# B&R Automation Studio project 8238 (part 6)

#### _config.st - *Read/Write Config Data
```iecst
ACTION _config:

	state 		ACCESS ADR(fuse.Internal.config_state);
	read_8		ACCESS ADR(fuse.Functions.Read_8);
	read_16		ACCESS ADR(fuse.Functions.Read_16);
	write		ACCESS ADR(fuse.Functions.Write);
	error		ACCESS ADR(fuse.Internal.LastError);

	read_8.pDeviceName 		:= fuse.pDevice;
	read_8.pData			:= ADR(fuse.Internal.Data_8);
	read_8.datatype 		:= ioLinkTYPE_USINT;
	read_8.dataLen			:= SIZEOF(fuse.Internal.Data_8);
	read_8.subIndex 		:= 0;

	read_16.pDeviceName 	:= fuse.pDevice;
	read_16.pData			:= ADR(fuse.Internal.Data_16);
	read_16.datatype 		:= ioLinkTYPE_UINT;
	read_16.dataLen			:= SIZEOF(fuse.Internal.Data_16);
	read_16.subIndex 		:= 0;

	write.pDeviceName := fuse.pDevice;
	write.pData 	:= ADR(fuse.Internal.WriteData);

	CASE state OF
		0:// Init  Turn of all functions just in case.
			fuse.Info.CommsOk := 0;
			state := 1;

		1://
			read_8.enable 	:= 0;
			read_8();
			IF (read_8.status = ERR_FUB_ENABLE_FALSE) THEN
				state := 2;
			END_IF;

		2:
			read_16.enable 	:= 0;
			read_16();
			IF (read_16.status = ERR_FUB_ENABLE_FALSE) THEN
				state := 3;
			END_IF;

		3..9:
			write.enable := 0;
			write();
			IF (write.status = ERR_FUB_ENABLE_FALSE) THEN
				state := 10;
			END_IF;

		10://Read the number of nodes.
			read_8.enable 	:= 1;
			read_8.index		:= 91;
			read_8();
			IF (read_8.status = ERR_OK) THEN
				fuse.Info.CommsOk := 1;
				fuse.Info.NoNodes := fuse.Internal.Data_8;
				fuse.Internal.Data_8 := 0;
				IF (fuse.Info.NoNodes > 0) THEN
					IF fuse.Info.NoNodes > MAX_FUSE_CHANNELS THEN
						fuse.Info.NoNodes := MAX_FUSE_CHANNELS;
					END_IF;
					state := 11;
				ELSE
					state := 0;
				END_IF;
			ELSIF (read_8.status <> ERR_FUB_BUSY) AND (read_8.status <> ERR_FUB_ENABLE_FALSE)  THEN  // Error read_8ing re initialise
				error := read_8.status;
				fuse.Info.CommsOk := 0;
				state := 0;
			END_IF;

		11..50:// read_8 the type  MAX 40 Fuses.
			channel := (state - 10);
			IF channel <= fuse.Info.NoNodes THEN
				read_8.enable 	:= 1;
				read_8.index		:= 900 + channel;
				read_8();
				IF (read_8.status = ERR_OK) THEN
					fuse.Info.Channel[channel].Type := fuse.Internal.Data_8;
					state := state + 1;
				ELSIF (read_8.status <> ERR_FUB_BUSY) AND (read_8.status <> ERR_FUB_ENABLE_FALSE)  THEN  // Error read_8ing re initialise
					fuse.Info.CommsOk := 0;
					state := 0;
				END_IF;
			ELSE
				state := 51;
			END_IF;

		51..90:// read_8 the trip current
			channel := (state - 50);
			IF channel <= fuse.Info.NoNodes THEN
				read_8.enable 	:= 1;
				read_8.index		:= 400 + channel;
				read_8();
				IF (read_8.status = ERR_OK) THEN
					fuse.Info.CommsOk := 1;
					fuse.Info.Channel[channel].TripCurrent := fuse.Internal.Data_8;
					state := state + 1;
				ELSIF (read_8.status <> ERR_FUB_BUSY) AND (read_8.status <> ERR_FUB_ENABLE_FALSE)  THEN  // Error reading re initialise
					state := 0;
				END_IF;
			ELSE
				state := 91;
			END_IF;

		91://Release the function block
			read_8.enable := 0;
			read_8();
			IF (read_8.status = ERR_FUB_ENABLE_FALSE) THEN
				state := 92;
			END_IF;

		92..93: // Read the max voltage
			read_16.enable := 1;
			read_16.datatype := ioLinkTYPE_INT;
			read_16.index		:= 100;
			read_16();
			IF (read_16.status = ERR_OK) THEN
				fuse.Info.CommsOk := 1;
				fuse.Info.MaxVoltage := fuse.Internal.Data_16;
				state := state + 1;
			ELSIF (read_16.status <> ERR_FUB_BUSY) AND (read_16.status <> ERR_FUB_ENABLE_FALSE)  THEN  // Error read_16ing re initialise
				fuse.Info.CommsOk := 0;
				state := 0;
			END_IF;

		94:// Read the Min Voltage;
			read_16.enable 	:= 1;
			read_16.datatype := ioLinkTYPE_INT;
			read_16.index		:= 101;
			read_16();
			IF (read_16.status = ERR_OK) THEN
				fuse.Info.CommsOk := 1;
				fuse.Info.MinVoltage :=  fuse.Internal.Data_16;
				state := state + 1;
			ELSIF (read_16.status <> ERR_FUB_BUSY) AND (read_16.status <> ERR_FUB_ENABLE_FALSE)  THEN  // Error reading re initialise
				fuse.Info.CommsOk := 0;
				state := 0;
			END_IF;

		95..100: // Disable the 16 way
			read_16.enable := 0;
			read_16();
			IF (read_16.status = ERR_FUB_ENABLE_FALSE) THEN
				state := 101;
			END_IF;

		101..140: // Read the channel status
			channel := (state - 100);
			IF channel <= fuse.Info.NoNodes THEN
				read_8.enable := 1;
				read_8.index := 500 + channel;
				read_8();
				IF (read_8.status = ERR_OK) THEN
					fuse.Info.Channel[channel].Status := fuse.Internal.Data_8;
					state := state + 1;
				END_IF;
			ELSE
				state := 141;
			END_IF;

		141: // Decide what to do next?
			//Check for differences then write if required
			//Check if the Min voltage has changed.
			IF (fuse.Info.MinVoltage <> fuse.Settings.MinVoltage) AND (fuse.Settings.MinVoltage > 0) THEN
				state := 150;
			END_IF;
			//Check if the Max voltage has changed.
			IF (fuse.Info.MaxVoltage <> fuse.Settings.MaxVoltage) AND (fuse.Settings.MaxVoltage > 0) THEN
				state := 151;
			END_IF;
			IF (fuse.Info.NoNodes > 0) THEN
				// Check if the trip current has changed
				FOR n := 1 TO fuse.Info.NoNodes DO
					IF (fuse.Info.Channel[n].TripCurrent <> fuse.Settings.Channel[n].TripCurrent) AND (fuse.Settings.Channel[n].TripCurrent > 0) THEN
						state := 161;
						EXIT;
					END_IF;
				END_FOR;
				// Check if the state has changed
				FOR n := 1 TO fuse.Info.NoNodes DO
					CASE fuse.Info.Channel[n].Status  OF
						EB_STATE_NC, EB_STATE_TRIP_SW_OFF:  // We cannot do anything is software.
							// We can;t do anything.

						EB_STATE_ON,EB_STATE_I_90, EB_STATE_I_100:
							IF (fuse.Settings.Channel[n].SetState = EB_SET_STATE_OFF ) THEN
								state := 200 + n;
								EXIT;
							END_IF;

						EB_STATE_TRIP, EB_STATE_TRIP_THERMAL, EB_STATE_TRIP_HARDWARE:
							IF (fuse.Settings.Channel[n].SetState = EB_SET_STATE_RESET ) THEN
								state := 200 + n;
								EXIT;
							END_IF;

						EB_STATE_OFF: // Turned off by hand
							IF (fuse.Settings.Channel[n].SetState = EB_SET_STATE_ON ) THEN
								state := 200 + n;
								EXIT;
							END_IF;
					END_CASE;
					IF (state = 141) THEN
						fuse.Settings.Channel[n].SetState := 0;	// Setting is not valid and cannot be actioned so clear it.
					END_IF;
				END_FOR;

				IF (state = 141) THEN
					state := 101;
				END_IF;

			ELSE
				state := 0;
			END_IF;

		142: // Disable the write FUB	AND read all the settings again.
			write.enable := 0;
			write();
			IF (write.status = ERR_FUB_ENABLE_FALSE) THEN
				state := 0;
			END_IF;

		150:// Write the Min Voltage
			fuse.Internal.WriteData := fuse.Settings.MinVoltage;
			write.enable := (fuse.Internal.WriteData > 0);
			write.index := 101;
			write.dataLen := 2;
			write.datatype := ioLinkTYPE_UINT;
			write();
			IF write.status = ERR_OK THEN
				state := 142;
			ELSIF (write.status < ERR_FUB_ENABLE_FALSE) THEN
				state := 0;
			ELSIF (fuse.Internal.WriteData = 0) THEN
				state := 142;
			END_IF;

		151:// Write the Max Voltage
			fuse.Internal.WriteData := fuse.Settings.MaxVoltage;
			write.enable := (fuse.Internal.WriteData > 0);
			write.index := 100;
			write.dataLen := 2;
			write.datatype := ioLinkTYPE_UINT;
			write();
			IF write.status = ERR_OK THEN
				state := 142;
			ELSIF (write.status < ERR_FUB_ENABLE_FALSE) THEN
				error := write.status;
				state := 0;
			ELSIF (fuse.Internal.WriteData = 0) THEN
				state := 142;
			END_IF;

		161..200:// Write the trip current current
			writeChannel := (state - 160);
			IF writeChannel > fuse.Info.NoNodes THEN
				state := 142;
			ELSE
				fuse.Internal.WriteData := fuse.Settings.Channel[writeChannel].TripCurrent;
				write.enable := (fuse.Internal.WriteData > 0);
				write.index := 400 + writeChannel;
				write.datatype := ioLinkTYPE_USINT;
				write.dataLen := 1;
				write();
				IF (write.status = ERR_OK) THEN
					state := state + 1;
				ELSIF (write.status = ERR_FUB_ENABLE_FALSE) THEN // Nothing to do
					state := state + 1;
				ELSIF (write.status <> ERR_FUB_BUSY) THEN
					error := write.status;
					state := 0;
				END_IF;
			END_IF;

		201..240:// Write the state.
			writeChannel := (state - 200);
			IF writeChannel > fuse.Info.NoNodes THEN
				state := 142;
			ELSE
				CASE fuse.Settings.Channel[writeChannel].SetState OF  // Manual setting of state.
					0: // Do nothing
						fuse.Internal.WriteData := 0;
					EB_SET_STATE_ON:// Digital ON  -- This will not override a push button OFF
						fuse.Internal.WriteData := ((writeChannel - 1) * 5) + 1;
					EB_SET_STATE_OFF:// Digital OFF
						fuse.Internal.WriteData := ((writeChannel - 1) * 5) + 2;
					EB_SET_STATE_RESET:// Reset
						fuse.Internal.WriteData := ((writeChannel - 1) * 5) + 3;
				END_CASE;
				write.enable := (fuse.Internal.WriteData > 0);
				write.index := 80;
				write.datatype := ioLinkTYPE_USINT;
				write.dataLen := 1;
				write();
				IF (write.status = ERR_OK) THEN
					fuse.Settings.Channel[writeChannel].SetState := 0;
					state := 142;
				ELSIF (write.status = ERR_FUB_ENABLE_FALSE) THEN // Nothing to do
					state := 142;
				ELSIF (write.status <> ERR_FUB_BUSY) THEN
					error := write.status;
					state := 0;
				ELSIF (fuse.Internal.WriteData = 0) THEN
					state := 142;
				END_IF;
			END_IF;

	END_CASE;

END_ACTION
```

#### _visuRead.st
```iecst
ACTION _visuRead:

	IF (index < 1 ) OR (index > MAX_FUSE_BANKS) THEN
		index := 1;
	END_IF;
	IF (visu_index < 1 ) THEN
		visu_index := MAX_FUSE_BANKS;
	ELSIF(visu_index > MAX_FUSE_BANKS) THEN
		visu_index := 1;
	END_IF;

	visu_fuse ACCESS ADR(Fuse[index]);
	visu_settings ACCESS ADR(gSettings.Fuse[index]);

	IF (visu_index <> last_visu_index) AND (visu_index > 0) THEN
		//Initialise visu settings.
		FOR n := 1 TO MAX_FUSE_CHANNELS DO
			brsitoa(gSettings.Fuse[visu_index].Channel[n].TripCurrent,ADR(visu_set_current[n]));
		END_FOR;
		last_visu_index := visu_index;
	ELSIF (visu_index = 0) THEN
		last_visu_index := 0;
	END_IF;

	readVoltage.pDeviceName := readCurrent.pDeviceName  := visu_fuse.pDevice;

	readVoltage.enable := 1;
	readVoltage.subIndex := readCurrent.subIndex :=  0;
	readVoltage.datatype := readCurrent.datatype := ioLinkTYPE_UINT;
	readVoltage.pData		:= ADR(inputVoltage);
	readVoltage.dataLen	:= SIZEOF(inputVoltage);
	readVoltage.index := 90;
	readVoltage();
	visu_fuse.Info.InputVoltage := inputVoltage;

	IF (act_current_channel < 1) THEN
		act_current_channel := 1;
	END_IF;

	//Cycle through the channel data
	readCurrent.enable := (act_current_channel <= visu_fuse.Info.NoNodes);
	readCurrent.pData		:= ADR(actualCurrent);
	readCurrent.dataLen	:= SIZEOF(actualCurrent);
	readCurrent.index := 300 + act_current_channel;
	readCurrent();
	IF (readCurrent.status = ERR_OK) THEN
		visu_fuse.Info.Channel[act_current_channel].ActualCurrent := actualCurrent;  // Scale the value here so we can see it correctly on the UI.
		act_current_channel := act_current_channel + 1;
	ELSIF (readCurrent.status = ERR_FUB_ENABLE_FALSE) THEN
		IF (visu_index > 0) AND (visu_index <= MAX_FUSE_BANKS)  THEN
			index := visu_index;
		ELSE
			index := index + 1;
		END_IF;
		act_current_channel := 1;
	ELSIF (readCurrent.status <> ERR_FUB_BUSY) THEN	 //ERROR try the next fuse
		visu_fuse.Info.Channel[act_current_channel].ActualCurrent := 100;//16#FFFF;  // Error value
		act_current_channel := act_current_channel + 1;
	END_IF;

	IF (visu_fuse.Info.NoNodes > 0) AND (index = visu_index) AND (visu_index > 0) THEN
		FOR n := 1 TO visu_fuse.Info.NoNodes DO
			CASE visu_fuse.Info.Channel[n].Status OF
				EB_STATE_NC, EB_STATE_TRIP_SW_OFF, EB_STATE_TRIP_HARDWARE: // Fuse failed: // Turned off by hand: // Not connected
					visu_action[n].Visible := 0;
					visu_action[n].visu_style := 'Kg_Red';

				EB_STATE_OFF:
					visu_action[n].Visible := 1;
					visu_action[n].Text  	:= '$$Fuses.Action.TurnOn';
					visu_action[n].visu_style := 'Kg_Red';
					IF visu_action[n].Value THEN
						visu_settings.Channel[n].SetState := EB_SET_STATE_ON;
						visu_action[n].Value := 0;
					END_IF;

				EB_STATE_ON, EB_STATE_I_90, EB_STATE_I_100:
					visu_action[n].Visible := 1;
					visu_action[n].Text  	:= '$$Fuses.Action.TurnOff';
					visu_action[n].visu_style := 'KannegiesserBlue';
					IF visu_action[n].Value THEN
						visu_settings.Channel[n].SetState := EB_SET_STATE_OFF;
						visu_action[n].Value := 0;
					END_IF;

				EB_STATE_TRIP,EB_STATE_TRIP_THERMAL:
					visu_action[n].Visible := 1;
					visu_action[n].Text  	:= '$$Fuses.Action.Reset';
					visu_action[n].visu_style := 'Kg_Orange';
					IF visu_action[n].Value THEN
						visu_settings.Channel[n].SetState := EB_SET_STATE_RESET;
						visu_action[n].Value := 0;
					END_IF;
			END_CASE;

			visu_settings.Channel[n].TripCurrent := DINT_TO_USINT(brsatoi(ADR(visu_set_current[n])));
		END_FOR
	END_IF;

	// We should clear the UI. if we are not reading correctly.
	IF (visu_index <> index) THEN
		visu_fuse.Info.CommsOk := 0;
	END_IF;

END_ACTION
```

#### Types.typ - Local data types
```iecst
(*Insert your comment here.*)

TYPE
	Fuse_typ : 	STRUCT
		Info : Fuse_Info_typ;
		Functions : FuseFunctions_typ;
		pDevice : UDINT; (**pointer to Address on IO Link interface*)
		Settings : FuseSetting_typ;
		Internal : FuseInternal_typ;
	END_STRUCT;
	Fuse_Info_typ : 	STRUCT  (*Actual Values Being read from the fuse*)
		CommsOk : BOOL; (*Comms Is Healthy*)
		NoNodes : USINT; (*91 - 8bit RO*)
		MinVoltage : INT; (*101 - 16Bit  R/W*)
		MaxVoltage : INT; (*100 - 16Bit  R/W*)
		InputVoltage : UINT;
		Channel : ARRAY[1..MAX_FUSE_CHANNELS]OF FuseChannel_Info_typ;
	END_STRUCT;
	FuseChannel_Info_typ : 	STRUCT
		Type : FuseType_enum;
		Status : FuseStatus_enum;
		TripCurrent : USINT;
		ActualCurrent : UINT;
	END_STRUCT;
	FuseType_enum :
		(
		EB_UNKNOWN := 0,
		EB_3824_100_0 := 170,
		EB_0824_100_0 := 138,
		EB_1824_010_0 := 145,
		EB_1824_020_0 := 146,
		EB_1824_030_0 := 147,
		EB_1824_040_0 := 148,
		EB_1824_060_0 := 150,
		EB_1824_080_0 := 152,
		EB_1824_100_0 := 154
		);
END_TYPE

(*Split up the function blocks, so we can read multiple pieces of data at once.*)

TYPE
	FuseFunctions_typ : 	STRUCT
		Read_8 : ioLinkRead; (*Read 8 bit register*)
		Read_16 : ioLinkRead; (*Read 16 register*)
		Write : ioLinkWrite;
	END_STRUCT;
	FuseInternal_typ : 	STRUCT  (*Internal bits for use*)
		config_state : UINT;
		LastError : UINT;
		Data_8 : USINT;
		Data_16 : UINT;
		WriteData : UINT;
	END_STRUCT;
	FuseStatus_enum :
		(
		EB_STATE_NC := 0, (*Not connected*)
		EB_STATE_OFF := 1, (*Switched Off - via software resetable*)
		EB_STATE_ON := 2, (*Switch On*)
		EB_STATE_TRIP := 3, (*Tripped*)
		EB_STATE_I_90 := 6, (*Current Exceeds 90%*)
		EB_STATE_I_100 := 14, (*Current Exceeds 100%*)
		EB_STATE_TRIP_HARDWARE := 18, (*Tripped - Hardware Error*)
		EB_STATE_TRIP_THERMAL := 20, (*Tripped - Thermal Release*)
		EB_STATE_TRIP_SW_OFF := 50 (*Switched Off Via the Button -- Cannot be overridden*)
		);
	visu_action_btn_typ : 	STRUCT
		Visible : BOOL;
		Text : STRING[25];
		Value : BOOL;
		visu_style : STRING[20] := 'KannegiesserBlue';
	END_STRUCT;
END_TYPE
```

#### Variables.var - Local variables
```iecst
VAR
	visu_fuse : REFERENCE TO Fuse_typ;
	Fuse : ARRAY[0..MAX_FUSE_BANKS] OF Fuse_typ;
	fuseTrippedAlarm : ARRAY[1..MAX_FUSE_BANKS] OF BOOL; (*alarm : REFERENCE TO Alm;*)
	reset : ARRAY[0..2] OF BOOL;
	fuseFault : ARRAY[0..2] OF BOOL;
	fuse : REFERENCE TO Fuse_typ;
	n : INT;
	plc : USINT;
	state : REFERENCE TO UINT;
	Channel : REFERENCE TO UINT;
	i : USINT;
	error : REFERENCE TO UINT;
	read_8 : REFERENCE TO ioLinkRead;
	read_16 : REFERENCE TO ioLinkRead;
	write : REFERENCE TO ioLinkWrite;
	channel : UINT;
	writeChannel : UINT;
	readVoltage : {REDUND_UNREPLICABLE} ioLinkRead;
	readCurrent : {REDUND_UNREPLICABLE} ioLinkRead;
	visu_index : USINT;
	act_current_channel : USINT;
	actualCurrent : UINT;
	inputVoltage : UINT;
	index : USINT;
	visu_settings : REFERENCE TO FuseSetting_typ;
	visu_action : ARRAY[0..MAX_FUSE_CHANNELS] OF visu_action_btn_typ;
	visu_set_current : ARRAY[0..MAX_FUSE_CHANNELS] OF STRING[3];
	last_visu_index : USINT;
	sIndex : STRING[5];
END_VAR
```

### Constants.var - Exported constants
```iecst
VAR CONSTANT
	CONTACTRON_CURRENT_STATUS : USINT := 15;
	CONTACTRON_WRITE_CURRENT : USINT := 128;
	CONTACTRON_TRIP_STATUS : USINT := 112;
	CONTACTRON_MAINS_LOSS : USINT := 32;
	CONTACTRON_PHASE_LOSS : USINT := 64;
END_VAR
(**Trip current Constants*)
VAR CONSTANT
	CONTACTRON_TRIP_MIN : USINT := 2#00000001; (*Overload current must be set in % in 15 increments*)
	CONTACTRON_TRIP_50_PERCENT : USINT := 2#00000111;
	CONTACTRON_TRIP_75_PERCENT : USINT := 2#00001100;
	CONTACTRON_TRIP_MAX : USINT := 2#00001111;
END_VAR
```

### IOlink.typ - Exported data types
```iecst
TYPE
	contactron_visu_manual_typ : 	STRUCT
		Visible : BOOL; (**Are the controls Visible*)
		Name : STRING[10];
		RunReverse : BOOL;
		RunForwards : BOOL;
		SetCurrent : INT;
		Error : BOOL;
		ErrorReset : BOOL;
		selectedIndex : UINT;
		selectedValue : STRING[10];
		refreshDropDown : R_TRIG;
		ListBoxVisible : BOOL;
		EnableRunReverse : BOOL;
		EnableRunForwards : BOOL;
		Enable : BOOL;
		Status : Contactron_Status_Type;
		ErrorString : STRING[400];
	END_STRUCT;
	contactron_manual_typ : 	STRUCT
		RunReverse : BOOL;
		RunForwards : BOOL;
		Enable : BOOL;
		ErrorReset : BOOL;
	END_STRUCT;
	Contactron_Cmd_Type : 	STRUCT
		Reset_Manual : BOOL;
		Reset_Automatic : BOOL;
		Stop : BOOL;
		Run : BOOL;
		Direction : Contactron_Direction;
		Current : USINT; (*Sets the trip current, enable must be off to write*)
	END_STRUCT;
	Contactron_Comms_Type : 	STRUCT
		Write : Contactron_Outputs_Type;
		Read : Contactron_Inputs_Type;
	END_STRUCT;
	Contactron_Device_Type :
		(
		CONTACTRON_H5_3 := 0,
		CONTACTRON_H5_9 := 1,
		CONTACTRON_H3_3 := 2,
		CONTACTRON_H3_9 := 3
		);
	Contactron_Direction :
		(
		CONTACTRON_FORWARD := 0,
		CONTACTRON_REVERSE := 1
		);
	Contactron_Inputs_Type : 	STRUCT
		Diagnostics : USINT;
		CurrentStatus : USINT; (*Current trip level and trip status*)
		ThermalPercentOfMax : USINT;
		CurrentPercentOfMax : USINT;
		DeviceType : USINT; (*Type of contactron used*)
		CurrentActual : USINT; (*10mA*)
		Data : ARRAY[0..7]OF USINT;
	END_STRUCT;
	Contactron_Outputs_Type : 	STRUCT
		Control : USINT;
		NominalCurrent : USINT;
	END_STRUCT;
	Contactron_Status_Type : 	STRUCT
		Error : BOOL;
		STO_Active : BOOL;
		Running : BOOL;
		Overload_Warning : BOOL;
		MainsFailure : BOOL;
		PhaseLoss : BOOL;
		Current : REAL;
		DeviceType : Contactron_Device_Type;
	END_STRUCT;
	Contactron_Type : 	STRUCT  (*Parent structure to hold all Contactron structures*)
		Cmd : Contactron_Cmd_Type;
		Status : Contactron_Status_Type;
		Comms : Contactron_Comms_Type;
		Manual : contactron_manual_typ;
	END_STRUCT;
	IO_Link_Type : 	STRUCT  (*Parent structure to hold all IO_Link device structures*)
		Contactron : ARRAY[0..MAX_CONTACTRON]OF Contactron_Type; (*Parent structure to hold all Contactron structures*)
	END_STRUCT;
END_TYPE

(**)

TYPE
	contactron_setting_typ : 	STRUCT
		Name : STRING[50];
		SetCurrent : INT;
	END_STRUCT;
END_TYPE
```

### Program Logical/Standard/IOLink/Contactron/Contactron (IEC, version 2.00.1)

#### Main.st - Init, cyclic, exit code
```iecst
(********************************************************************
 * COPYRIGHT --
 ********************************************************************
 * PROGRAM: IOLink
 * File: IOLink_Driver.s
 * Author: Stephen Healy NOT ANYMORE :)
 * Created: Sept 05, 2018
 ********************************************************************
 * Implementation OF PROGRAM IOLink
 ********************************************************************)
//V1.00.1 First Release
//V1.00.1 TR 10/11/2020  - Remove run signal from contactron when there is a fault to allow the error to be acknowledged.
//V1.00.2 TR 07/04/2021  - Add Test mode

//V2.00.1 -- Remove dependency on shitty firmware hack- Add mappview visu support

PROGRAM _INIT

END_PROGRAM

PROGRAM _CYCLIC

	//Call contactron action
	IF MAX_CONTACTRON > 0 THEN
		_visu;
		_Contactron;

	END_IF;

END_PROGRAM
```

#### Variables.var - Local variables
```iecst
VAR
	n : UINT;
END_VAR
VAR CONSTANT
	max_manualControls : USINT := 8;
END_VAR
VAR
	visu_man : REFERENCE TO contactron_visu_manual_typ;
	visu_manual : ARRAY[0..max_manualControls] OF contactron_visu_manual_typ;
	selIndex : DINT;
	updateDropDown : BOOL;
	index : UINT;
	manualSelectDrowDown : ARRAY[0..MAX_CONTACTRON] OF STRING[125];
	sIndex : STRING[10];
	run : BOOL;
	contactron : REFERENCE TO Contactron_Type;
	RunMotor : BOOL;
	name : STRING[30];
END_VAR
VAR CONSTANT
	CONTACTRON_MANUAL_DEFAULT : contactron_manual_typ := (RunReverse:=0,RunForwards:=0,Enable:=0,ErrorReset:=0);
END_VAR
VAR
	errorString : STRING[400];
END_VAR
```

#### _Contactron.st
```iecst
ACTION _Contactron:
	//----------------------------------------------
	//-----------------Contactron-------------------
	//----------------------------------------------

	//Write control word
	FOR n:=1 TO MAX_CONTACTRON DO
		contactron ACCESS ADR(IO_Link.Contactron[n]);

		IF Std.TestMode  THEN
			contactron.Status.Running := 1;
			IF contactron.Cmd.Run THEN
				contactron.Status.Current := 1.0;
			ELSE
				contactron.Status.Current := 0.0;
			END_IF;

		ELSE
			brsmemcpy(ADR(contactron.Comms.Read.CurrentActual) + 1,ADR(contactron.Comms.Read.Data[1]),1);//High Byte
			brsmemcpy(ADR(contactron.Comms.Read.CurrentActual),ADR(contactron.Comms.Read.Data[2]),1);// Low Byte
			contactron.Comms.Read.DeviceType 			:= contactron.Comms.Read.Data[3];//2
			contactron.Comms.Read.ThermalPercentOfMax 	:= contactron.Comms.Read.Data[4];//3
			contactron.Comms.Read.CurrentPercentOfMax 	:= contactron.Comms.Read.Data[5];//4
			contactron.Comms.Read.CurrentStatus 		:= contactron.Comms.Read.Data[6];//5
			contactron.Comms.Read.Diagnostics 			:= contactron.Comms.Read.Data[7];//6

			//Read status
			contactron.Status.Error 			:= contactron.Comms.Read.Diagnostics.0;
			contactron.Status.STO_Active 		:= NOT contactron.Comms.Read.Diagnostics.3;
			contactron.Status.Running 		:= contactron.Comms.Read.Diagnostics.5;
			contactron.Status.Overload_Warning 	:= contactron.Comms.Read.Diagnostics.6;
			contactron.Status.MainsFailure 		:= ((contactron.Comms.Read.CurrentStatus AND CONTACTRON_TRIP_STATUS) = CONTACTRON_MAINS_LOSS);
			contactron.Status.PhaseLoss 		:= ((contactron.Comms.Read.CurrentStatus AND CONTACTRON_TRIP_STATUS) = CONTACTRON_PHASE_LOSS);
			contactron.Status.Current 			:= contactron.Comms.Read.CurrentActual * 0.01;
			contactron.Status.DeviceType 		:= contactron.Comms.Read.DeviceType;

			IF contactron.Status.Error THEN
				run := 0;
			ELSIF contactron.Manual.Enable THEN
				run := 0;
				contactron.Comms.Write.Control.0 := contactron.Manual.RunForwards;
				contactron.Comms.Write.Control.7 := contactron.Manual.RunForwards;
				contactron.Comms.Write.Control.1 := contactron.Manual.RunReverse;
				contactron.Comms.Write.Control.5 := contactron.Manual.RunReverse;
			ELSE
				run := contactron.Cmd.Run;
			END_IF;

			IF NOT 	contactron.Manual.Enable THEN

				CASE contactron.Cmd.Direction OF
					CONTACTRON_FORWARD:
						contactron.Comms.Write.Control.0 := run;
						contactron.Comms.Write.Control.7 := run;
						contactron.Comms.Write.Control.1 := FALSE;
						contactron.Comms.Write.Control.5 := FALSE;

					CONTACTRON_REVERSE:
						contactron.Comms.Write.Control.0 := FALSE;
						contactron.Comms.Write.Control.7 := FALSE;
						contactron.Comms.Write.Control.1 := run;
						contactron.Comms.Write.Control.5 := run;

					ELSE
						contactron.Comms.Write.Control.0 := FALSE;
						contactron.Comms.Write.Control.7 := FALSE;
						contactron.Comms.Write.Control.1 := FALSE;
						contactron.Comms.Write.Control.5 := FALSE;
				END_CASE;
			END_IF;
			contactron.Comms.Write.Control.2 := contactron.Cmd.Reset_Manual OR contactron.Manual.ErrorReset;
			contactron.Comms.Write.Control.3 := contactron.Cmd.Reset_Automatic;
			contactron.Comms.Write.Control.4 := FALSE; //NOT USED
			contactron.Comms.Write.Control.6 := contactron.Cmd.Stop;

			IF contactron.Cmd.Current > 0 THEN //Write trip current level
				contactron.Comms.Write.NominalCurrent := (contactron.Cmd.Current OR CONTACTRON_WRITE_CURRENT);
			ELSE
				contactron.Comms.Write.NominalCurrent := 0;
			END_IF;
			IF contactron.Cmd.Current = (contactron.Comms.Read.CurrentStatus AND CONTACTRON_CURRENT_STATUS) THEN
				contactron.Cmd.Current := 0; //Reset trip current if cmd written
			END_IF;

		END_IF;

		//Clear the manual commands.
		contactron.Manual := CONTACTRON_MANUAL_DEFAULT;
	END_FOR;
END_ACTION
```

#### _visu.st
```iecst
ACTION _visu:

	FOR n := 1 TO max_manualControls DO

		visu_man ACCESS ADR(visu_manual[n]);

		selIndex := atoi(ADR(visu_man.selectedValue));
		IF (selIndex > 0) AND (selIndex <= MAX_CONTACTRON) AND (selIndex <> visu_man.selectedIndex) THEN
			updateDropDown := 1;
			visu_man.selectedIndex := DINT_TO_UINT(selIndex);
		END_IF;

		visu_man.ListBoxVisible := (visu_man.selectedIndex = 0);

		visu_man.refreshDropDown.CLK := (visu_man.selectedIndex = 0);
		visu_man.refreshDropDown();
		IF visu_man.refreshDropDown.Q THEN
			updateDropDown := 1;
		END_IF;

		contactron ACCESS ADR(IO_Link.Contactron[visu_man.selectedIndex]);
		contactron.Manual.Enable := 1; //Mark Contactron as in manual mode

		visu_man.Visible 		:= (visu_man.selectedIndex > 0);
		IF (gSettings.Contactron[visu_man.selectedIndex].Name <> '') THEN
			visu_man.Name    		:= gSettings.Contactron[visu_man.selectedIndex].Name;
		ELSE
			itoa(visu_man.selectedIndex,ADR(sIndex));
			visu_man.Name  := 'C ';
			brsstrcat(ADR(visu_man.Name ),ADR(sIndex));
		END_IF;

		visu_man.Status			 	:= contactron.Status;

		visu_man.Error := visu_man.Status.Error OR visu_man.Status.STO_Active OR visu_man.Status.Overload_Warning
											OR visu_man.Status.MainsFailure OR visu_man.Status.PhaseLoss;

		errorString := '';
		// We can;t use the text from the database as it doesn;t understand the end of line characters
		IF visu_man.Status.Error THEN
			brsstrcat(ADR(errorString),ADR('Error'));//brsstrcat(ADR(errorString),ADR('$$IAT/Contactron.Error'));
			brsstrcat(ADR(errorString),ADR('\n'));
		END_IF;
		IF visu_man.Status.STO_Active THEN
			brsstrcat(ADR(errorString),ADR('STO Active'));//brsstrcat(ADR(errorString),ADR('$$IAT/Contactron.STO'));
			brsstrcat(ADR(errorString),ADR('\n'));
		END_IF;
		IF visu_man.Status.Overload_Warning THEN
			brsstrcat(ADR(errorString),ADR('Overload Warning'));//brsstrcat(ADR(errorString),ADR('$$IAT/Contactron.Overload'));
			brsstrcat(ADR(errorString),ADR('\n'));
		END_IF;
		IF visu_man.Status.MainsFailure THEN
			brsstrcat(ADR(errorString),ADR('Mains Failure'));//brsstrcat(ADR(errorString),ADR('$$IAT/Contactron.MainsFailure'));
			brsstrcat(ADR(errorString),ADR('\n'));
		END_IF;
		IF visu_man.Status.PhaseLoss THEN
			brsstrcat(ADR(errorString),ADR('Phase Loss'));//brsstrcat(ADR(errorString),ADR('$$IAT/Contactron.PhaseLoss'));
		END_IF;

		brsstrcpy(ADR(visu_man.ErrorString),ADR(errorString));

		IF visu_man.ErrorReset THEN
			visu_man.ErrorReset := 0;
			contactron.Manual.ErrorReset := 1;
		END_IF;

		visu_man.Enable := NOT contactron.Status.Error;

		IF NOT visu_man.Enable THEN
			visu_man.RunReverse							:= 0;
			visu_man.RunForwards						:= 0;
			visu_man.EnableRunReverse   		:= 0;
			visu_man.EnableRunForwards			:= 0;
		ELSIF visu_man.RunForwards THEN
			contactron.Manual.RunForwards 	:= 1;
			visu_man.EnableRunReverse	  		:= 0;
		ELSIF visu_man.RunReverse THEN
			contactron.Manual.RunReverse		:= 1;
			visu_man.EnableRunForwards			:= 0;
		ELSE
			visu_man.EnableRunReverse				:= 1;
			visu_man.EnableRunForwards			:= 1;
		END_IF;

	END_FOR;

	//Build the list box string;
	//[{'value':'text_1', 'text':'$$IAT/testText1'}, {'value':'text_2', 'text':'$$IAT/testText2'}]
	IF updateDropDown THEN
		index := 1;
		brsmemset(ADR(manualSelectDrowDown),0,SIZEOF(manualSelectDrowDown));
		manualSelectDrowDown[0] := '{"value":0,"text":""}';
		FOR n := 1 TO MAX_CONTACTRON DO
			contactron ACCESS ADR(IO_Link.Contactron[n]);
			IF NOT contactron.Manual.Enable THEN
				itoa(n,ADR(sIndex));

				IF (gSettings.Contactron[n].Name <> '') THEN
					name := gSettings.Contactron[n].Name;
				ELSE
					name := 'C ';
					brsstrcat(ADR(name),ADR(sIndex));
				END_IF;
				brsstrcat(ADR(manualSelectDrowDown[index]),ADR('{"value":"'));
				brsstrcat(ADR(manualSelectDrowDown[index]),ADR(sIndex));
				brsstrcat(ADR(manualSelectDrowDown[index]),ADR('","text":"'));
				brsstrcat(ADR(manualSelectDrowDown[index]),ADR(name));
				brsstrcat(ADR(manualSelectDrowDown[index]),ADR('"}'));
				index := index + 1;
			END_IF;
		END_FOR;
		updateDropDown := FALSE;
	END_IF;

END_ACTION
```

### IOlink.typ - not listed in the package file held
```iecst
TYPE
	IO_Link_FuseSettings_type : 	STRUCT
		Contactron : ARRAY[0..MAX_CONTACTRON]OF USINT;
	END_STRUCT;
	IO_Link_Type : 	STRUCT  (*Parent structure to hold all IO_Link device structures*)
		Device : STRING[80]; (*Physical address of the X20DS438A port to be used for EasyB*)
		Contactron : ARRAY[0..MAX_CONTACTRON]OF Contactron_Type; (*Parent structure to hold all Contactron structures*)
		Status : BOOL;
	END_STRUCT;
	Contactron_Inputs_Type : 	STRUCT
		Diagnostics : USINT;
		CurrentStatus : USINT; (*Current trip level and trip status*)
		ThermalPercentOfMax : USINT;
		CurrentPercentOfMax : USINT;
		DeviceType : USINT; (*Type of contactron used*)
		CurrentActual : USINT; (*10mA*)
		Data : ARRAY[0..5]OF USINT;
	END_STRUCT;
	Contactron_Outputs_Type : 	STRUCT
		Control : USINT;
		NominalCurrent : USINT;
	END_STRUCT;
	Contactron_Cmd_Type : 	STRUCT
		Reset_Manual : BOOL;
		Reset_Automatic : BOOL;
		Stop : BOOL;
		Run : BOOL;
		Direction : Contactron_Direction;
		Current : USINT; (*Sets the trip current, enable must be off to write*)
	END_STRUCT;
	Contactron_Status_Type : 	STRUCT
		Error : BOOL;
		STO_Active : BOOL;
		Device_Ok : BOOL;
		Overload_Warning : BOOL;
		MainsFailure : BOOL;
		PhaseLoss : BOOL;
		Current : REAL;
		DeviceType : Contactron_Device_Type;
	END_STRUCT;
	Contactron_Comms_Type : 	STRUCT
		Write : Contactron_Outputs_Type;
		Read : Contactron_Inputs_Type;
	END_STRUCT;
	Contactron_Type : 	STRUCT  (*Parent structure to hold all Contactron structures*)
		Cmd : Contactron_Cmd_Type;
		Status : Contactron_Status_Type;
		Comms : Contactron_Comms_Type;
	END_STRUCT;
	Contactron_Device_Type :
		(
		CONTACTRON_H5_3 := 0,
		CONTACTRON_H5_9 := 1,
		CONTACTRON_H3_3 := 2,
		CONTACTRON_H3_9 := 3
		);
	Contactron_Direction :
		(
		CONTACTRON_FORWARD := 0,
		CONTACTRON_REVERSE := 1
		);
END_TYPE
```

### Constants.var - not listed in the package file held
```iecst
VAR CONSTANT
	EASYB_STATE_5 : USINT := 5;
	EASYB_TRIPPED : USINT := 3;
	EASYB_SWITCHED_ON : USINT := 2;
	CONTACTRON_CURRENT_STATUS : USINT := 15;
	CONTACTRON_WRITE_CURRENT : USINT := 128;
	CONTACTRON_TRIP_STATUS : USINT := 112;
	CONTACTRON_MAINS_LOSS : USINT := 32;
	CONTACTRON_PHASE_LOSS : USINT := 64;
END_VAR
(**Trip current Constants*)
VAR CONSTANT
	CONTACTRON_TRIP_MIN : USINT := 2#00000001; (*Overload current must be set in % in 15 increments*)
	CONTACTRON_TRIP_50_PERCENT : USINT := 2#00000111;
	CONTACTRON_TRIP_75_PERCENT : USINT := 2#00001100;
	CONTACTRON_TRIP_MAX : USINT := 2#00001111;
END_VAR
```

### IOLink.var - not listed in the package file held
```iecst
VAR
	IO_Link : IO_Link_Type;
	Fuse_PB_Reset : ARRAY[0..2] OF BOOL;
	Fuse_PB_Lamp : ARRAY[0..2] OF BOOL;
END_VAR
```

### Program Logical/Standard/IOLink/IOLink_Driver (IEC, version 1.00.1)

#### Main.st - Init, cyclic, exit code
```iecst
(********************************************************************
 * COPYRIGHT --
 ********************************************************************
 * PROGRAM: IOLink
 * File: IOLink_Driver.st
 * Author: Stephen Healey
 * Created: Sept 05, 2018
 ********************************************************************
 * Implementation OF PROGRAM IOLink
 ********************************************************************)
//V1.00.1 First Release
//V1.00.1 TR 10/11/2020  - Remove run signal from contactron when there is a fault to allow the error to be acknowledged.

//	Description
//IOLink task for controlling Contactron's and EasyB's
//Constants need to be set. MAX_CONTACTRON and MAX_EASYB should match the hardware
//IO needs to be mapped for the Contactron's in the X20DS438A
//EasyB's IO does not need mapping. The interface still needs enabling in the X20DS438A config

//-------------------------------------------------------------
//-----------------------------Init----------------------------
//-------------------------------------------------------------
//	1.	Configures IOLink physical device, adjust address as needed
//	2.	Resets the controller state, needs to start offset, not 0

//-------------------------------------------------------------
//-----------------------------Cyclic--------------------------
//-------------------------------------------------------------
//	1.	Calls contactron action only if MAX_CONTACTRON is greater than zero
//	2.	Calls easyB action only if MAX_EASYB is greater than zero
//	3.	Monitors tripped status of all the EasyB's and enables reseting

//Use the following charts when setting the trip currents for the IOLink devices

//Contactron 												EasyB
//Current Setting Chart							Current Setting Chart
//Bit 		Nominal current						Enum										USINT			Value
//3 2 1 0 [mA]																													[mA]
//				 3 A 9 A
//0 0 0 0 180 1500									TRIP_CURRENT_DEFAULT		0					N/A
//0 0 0 1 300 2000									TRIP_CURRENT_500mA			5					500
//0 0 1 0 440 2500									TRIP_CURRENT_1A					10				1000
//0 0 1 1 600 3000									TRIP_CURRENT_2A					20				2000
//0 1 0 0 680 3500									TRIP_CURRENT_3A					30				3000
//0 1 0 1 880 4000									TRIP_CURRENT_4A					40				4000
//0 1 1 0 1000 4500									TRIP_CURRENT_5A					50				5000
//0 1 1 1 1100 5000									TRIP_CURRENT_6A					60				6000
//1 0 0 0 1200 5500									TRIP_CURRENT_8A					80				8000
//1 0 0 1 1500 6000									TRIP_CURRENT_10A				100				10000
//1 0 1 0 1600 6500
//1 0 1 1 1900 7000
//1 1 0 0 2100 7500
//1 1 0 1 2400 8000
//1 1 1 0 2700 8500
//1 1 1 1 3000 9000

PROGRAM _INIT
	//Configuration

	//Reset state

	backUp.fileDevice := 'UserPart';
	backUp.filePath := 'FuseTripConfig';

	//Load from file on boot

	backUp.step := backUpOpen;
END_PROGRAM

PROGRAM _CYCLIC
	//Call status
	IF IO_Link.Status THEN
	 _status;
	END_IF;

	//Call httpResponse conditionally
//	IF IO_Link.Load THEN
//		_backUpRead;
//		_encodeData;
//	END_IF;

	//Call httpRequest conditionally
//	IF IO_Link.Save THEN
//		_decodeData;
//		_backUpWrite;
//		_encodeData;
//	END_IF;

	//Call contactron action
	IF MAX_CONTACTRON > 0 THEN
		_Contactron;
	END_IF;

//	//Call easy b action
//	IF (MAX_EASYB > 0) AND (MAX_EASYB <= 40) THEN
//		_EasyB;
//
//		//Monitor Tripped status
//		IO_Link.EasyB.Tripped := FALSE;
//		FOR n:=1 TO MAX_EASYB DO
//			IF IO_Link.EasyB.EasyB_Array[n].Status.TripState = EASYB_TRIPPED THEN
//				IO_Link.EasyB.Tripped := TRUE;
//				EXIT;
//			END_IF;
//		END_FOR;
//		//Reset Tripped status
//		IF IO_Link.EasyB.Tripped AND IO_Link.EasyB.Reset THEN
//			FOR n:=1 TO MAX_EASYB DO
//				IF IO_Link.EasyB.EasyB_Array[n].Status.TripState = EASYB_TRIPPED THEN
//					IO_Link.EasyB.EasyB_Array[n].Cmd.Reset := TRUE;
//				END_IF;
//			END_FOR;
//			IO_Link.EasyB.Reset := FALSE;
//		END_IF;
//		IO_Link.EasyB.TrippedLamp := IO_Link.EasyB.Tripped AND Std.Clock1s;
//	END_IF;

END_PROGRAM
```

#### Types.typ - Local data types
```iecst
TYPE
	state_enum :
		(
		CONTACTRON := 0,
		EASYB := 1
		);
	BackUp : 	STRUCT
		filePath : STRING[15];
		fileDevice : STRING[10];
		status : UINT;
		ident : UDINT;
		step : backUp_enum;
		functions : backUp_functions;
	END_STRUCT;
	backUp_enum :
		(
		backUpStart := 0,
		backUpOpen := 1,
		backUpCreate := 2,
		backUpWrite := 3,
		backUpRead := 4,
		backUpClose := 5,
		backUpErrorRead := 6,
		backUpErrorWrite := 7,
		backUpExit := 100
		);
	backUp_functions : 	STRUCT
		fWrite : FileWrite;
		fRead : FileRead;
		fOpen : FileOpen;
		fCreate : FileCreate;
		fClose : FileClose;
	END_STRUCT;
END_TYPE
```

#### Variables.var - Local variables
```iecst
VAR
	n : USINT;
	fuseSettingStructure : IO_Link_FuseSettings_type;
	openFile : FileOpen;
	readFile : FileRead;
	closeFile : FileClose;
	writeFile : FileWrite;
	offset : USINT;
	statusState : USINT;
	statusValue : ARRAY[0..49] OF REAL;
	tempString : STRING[10];
	backUp : BackUp;
	state : state_enum;
	count : USINT;
	loop : UINT;
	tempString2 : STRING[5];
END_VAR
```

#### _EasyB.st
```iecst
ACTION _EasyB:
	//----------------------------------------------
	//--------------------Easy-B--------------------
	//----------------------------------------------

	//Read Controller Data
	IO_Link.EasyB.ControllerRead.enable := TRUE;
	IO_Link.EasyB.ControllerRead.pDeviceName := ADR(IO_Link.Device);

	CASE IO_Link.EasyB.ControllerState OF
		EASYB_READ_NUMBER_OF_NODES:
			//Specific function config
			IO_Link.EasyB.ControllerRead.index := 91;
			IO_Link.EasyB.ControllerRead.subIndex := 0;
			IO_Link.EasyB.ControllerRead.pData := ADR(IO_Link.EasyB.ControllerNumberOfNodes);
			IO_Link.EasyB.ControllerRead.dataLen := SIZEOF(IO_Link.EasyB.ControllerNumberOfNodes);
			IO_Link.EasyB.ControllerRead.datatype := ioLinkTYPE_SINT;
			IO_Link.EasyB.ControllerRead();
			//Goto next state
			IF IO_Link.EasyB.ControllerRead.status <> ERR_FUB_BUSY THEN
				IO_Link.EasyB.ControllerState := EASYB_READ_SUPPLY_VOLTAGE;
			END_IF;

		EASYB_READ_SUPPLY_VOLTAGE:
			//Specific function config
			IO_Link.EasyB.ControllerRead.index := 90;
			IO_Link.EasyB.ControllerRead.subIndex := 0;
			IO_Link.EasyB.ControllerRead.pData := ADR(IO_Link.EasyB.ControllerSupplyVoltage);
			IO_Link.EasyB.ControllerRead.dataLen := SIZEOF(IO_Link.EasyB.ControllerSupplyVoltage);
			IO_Link.EasyB.ControllerRead.datatype := ioLinkTYPE_INT;
			IO_Link.EasyB.ControllerRead();
			//Goto next state
			IF IO_Link.EasyB.ControllerRead.status <> ERR_FUB_BUSY THEN
				IO_Link.EasyB.ControllerState := EASYB_READ_NUMBER_OF_NODES;
			END_IF;
	END_CASE;

	//----------------------------------------------
	//-----------------Read Fuse Data---------------
	//----------------------------------------------
	FOR n:=1 TO MAX_EASYB DO
		IO_Link.EasyB.EasyB_Array[n].Comms.Read.enable := TRUE;
		IO_Link.EasyB.EasyB_Array[n].Comms.Read.pDeviceName := ADR(IO_Link.Device);

		CASE IO_Link.EasyB.EasyB_Array[n].State OF
			EASYB_READ_CURRENT:
				//Specific function config
				IO_Link.EasyB.EasyB_Array[n].Comms.Read.index := 300 + n;
				IO_Link.EasyB.EasyB_Array[n].Comms.Read.subIndex := 0;
				IO_Link.EasyB.EasyB_Array[n].Comms.Read.pData := ADR(IO_Link.EasyB.EasyB_Array[n].Status.Current);
				IO_Link.EasyB.EasyB_Array[n].Comms.Read.dataLen := SIZEOF(IO_Link.EasyB.EasyB_Array[n].Status.Current);
				IO_Link.EasyB.EasyB_Array[n].Comms.Read.datatype := ioLinkTYPE_INT;
				IO_Link.EasyB.EasyB_Array[n].Comms.Read();
				//Goto next state
				IF IO_Link.EasyB.EasyB_Array[n].Comms.Read.status <> ERR_FUB_BUSY THEN
					IO_Link.EasyB.EasyB_Array[n].State := EASYB_READ_TRIPPED;
				END_IF;

			EASYB_READ_TRIPPED:
				//Specific function config
				IO_Link.EasyB.EasyB_Array[n].Comms.Read.index := 500 + n;
				IO_Link.EasyB.EasyB_Array[n].Comms.Read.subIndex := 0;
				IO_Link.EasyB.EasyB_Array[n].Comms.Read.pData := ADR(IO_Link.EasyB.EasyB_Array[n].Status.TripState);
				IO_Link.EasyB.EasyB_Array[n].Comms.Read.dataLen := 1;
				IO_Link.EasyB.EasyB_Array[n].Comms.Read.datatype := ioLinkTYPE_USINT;
				IO_Link.EasyB.EasyB_Array[n].Comms.Read();
				//Goto next state
				IF IO_Link.EasyB.EasyB_Array[n].Comms.Read.status <> ERR_FUB_BUSY THEN
					IO_Link.EasyB.EasyB_Array[n].State := EASYB_READ_TRIP_COUNT;
				END_IF;

			EASYB_READ_TRIP_COUNT:
				//Specific function config
				IO_Link.EasyB.EasyB_Array[n].Comms.Read.index := 200 + n;
				IO_Link.EasyB.EasyB_Array[n].Comms.Read.subIndex := 0;
				IO_Link.EasyB.EasyB_Array[n].Comms.Read.pData := ADR(IO_Link.EasyB.EasyB_Array[n].Status.TripCount);
				IO_Link.EasyB.EasyB_Array[n].Comms.Read.dataLen := SIZEOF(IO_Link.EasyB.EasyB_Array[n].Status.TripCount);
				IO_Link.EasyB.EasyB_Array[n].Comms.Read.datatype := ioLinkTYPE_USINT;
				IO_Link.EasyB.EasyB_Array[n].Comms.Read();
				//Goto next state
				IF IO_Link.EasyB.EasyB_Array[n].Comms.Read.status <> ERR_FUB_BUSY THEN
					IO_Link.EasyB.EasyB_Array[n].State := EASYB_READ_TRIP_CURRENT;
				END_IF;

			EASYB_READ_TRIP_CURRENT:
				//Specific function config
				IO_Link.EasyB.EasyB_Array[n].Comms.Read.index := 400 + n;
				IO_Link.EasyB.EasyB_Array[n].Comms.Read.subIndex := 0;
				IO_Link.EasyB.EasyB_Array[n].Comms.Read.pData := ADR(IO_Link.EasyB.EasyB_Array[n].Status.TripCurrent);
				IO_Link.EasyB.EasyB_Array[n].Comms.Read.dataLen := 1;
				IO_Link.EasyB.EasyB_Array[n].Comms.Read.datatype := ioLinkTYPE_USINT;
				IO_Link.EasyB.EasyB_Array[n].Comms.Read();
				//Goto next state
				IF IO_Link.EasyB.EasyB_Array[n].Comms.Read.status <> ERR_FUB_BUSY THEN
					IO_Link.EasyB.EasyB_Array[n].State := EASYB_READ_FUSE_TYPE;
				END_IF;

			EASYB_READ_FUSE_TYPE:
				//Specific function config
				IO_Link.EasyB.EasyB_Array[n].Comms.Read.index := 900 + n;
				IO_Link.EasyB.EasyB_Array[n].Comms.Read.subIndex := 0;
				IO_Link.EasyB.EasyB_Array[n].Comms.Read.pData := ADR(IO_Link.EasyB.EasyB_Array[n].Status.Type);
				IO_Link.EasyB.EasyB_Array[n].Comms.Read.dataLen := 1;
				IO_Link.EasyB.EasyB_Array[n].Comms.Read.datatype := ioLinkTYPE_USINT;
				IO_Link.EasyB.EasyB_Array[n].Comms.Read();
				//Goto next state
				IF IO_Link.EasyB.EasyB_Array[n].Comms.Read.status <> ERR_FUB_BUSY THEN
					IO_Link.EasyB.EasyB_Array[n].State := EASYB_READ_CURRENT;
				END_IF;
		END_CASE;

		//----------------------------------------------
		//-----------------Write Fuse Data--------------
		//----------------------------------------------
		IO_Link.EasyB.EasyB_Array[n].Comms.Write.enable := TRUE;
		IO_Link.EasyB.EasyB_Array[n].Comms.Write.pDeviceName := ADR(IO_Link.Device);

		//Use ELSIF statement so only one action can happen at once as dataToWrite is shared.
		IF IO_Link.EasyB.EasyB_Array[n].Cmd.On THEN
			//Specific function config
			IO_Link.EasyB.EasyB_Array[n].Comms.Write.index := 80;
			IO_Link.EasyB.EasyB_Array[n].Comms.Write.subIndex := 0;
			IO_Link.EasyB.EasyB_Array[n].Comms.dataToWrite := (1 + ((n-1)*5));
			IO_Link.EasyB.EasyB_Array[n].Comms.Write.pData := ADR(IO_Link.EasyB.EasyB_Array[n].Comms.dataToWrite);
			IO_Link.EasyB.EasyB_Array[n].Comms.Write.dataLen := 1;
			IO_Link.EasyB.EasyB_Array[n].Comms.Write.datatype := ioLinkTYPE_USINT;
			IO_Link.EasyB.EasyB_Array[n].Comms.Write();
			//Goto next state
			IF IO_Link.EasyB.EasyB_Array[n].Comms.Write.status <> ERR_FUB_BUSY THEN
				IO_Link.EasyB.EasyB_Array[n].Cmd.On := FALSE;
			END_IF;
		ELSIF IO_Link.EasyB.EasyB_Array[n].Cmd.Off THEN
			//Specific function config
			IO_Link.EasyB.EasyB_Array[n].Comms.Write.index := 80;
			IO_Link.EasyB.EasyB_Array[n].Comms.Write.subIndex := 0;
			IO_Link.EasyB.EasyB_Array[n].Comms.dataToWrite := (2 + ((n-1)*5));
			IO_Link.EasyB.EasyB_Array[n].Comms.Write.pData := ADR(IO_Link.EasyB.EasyB_Array[n].Comms.dataToWrite);
			IO_Link.EasyB.EasyB_Array[n].Comms.Write.dataLen := 1;
			IO_Link.EasyB.EasyB_Array[n].Comms.Write.datatype := ioLinkTYPE_USINT;
			IO_Link.EasyB.EasyB_Array[n].Comms.Write();
			//Goto next state
			IF IO_Link.EasyB.EasyB_Array[n].Comms.Write.status <> ERR_FUB_BUSY THEN
				IO_Link.EasyB.EasyB_Array[n].Cmd.Off := FALSE;
			END_IF;
		ELSIF IO_Link.EasyB.EasyB_Array[n].Cmd.Reset THEN
			//Specific function config
			IO_Link.EasyB.EasyB_Array[n].Comms.Write.index := 80;
			IO_Link.EasyB.EasyB_Array[n].Comms.Write.subIndex := 0;
			IO_Link.EasyB.EasyB_Array[n].Comms.dataToWrite := (3 + ((n-1)*5));
			IO_Link.EasyB.EasyB_Array[n].Comms.Write.pData := ADR(IO_Link.EasyB.EasyB_Array[n].Comms.dataToWrite);
			IO_Link.EasyB.EasyB_Array[n].Comms.Write.dataLen := 1;
			IO_Link.EasyB.EasyB_Array[n].Comms.Write.datatype := ioLinkTYPE_USINT;
			IO_Link.EasyB.EasyB_Array[n].Comms.Write();
			//Goto next state
			IF IO_Link.EasyB.EasyB_Array[n].Comms.Write.status <> ERR_FUB_BUSY THEN
				IO_Link.EasyB.EasyB_Array[n].Cmd.Reset := FALSE;
			END_IF;
		ELSIF IO_Link.EasyB.EasyB_Array[n].Cmd.ClearCounter THEN
			//Specific function config
			IO_Link.EasyB.EasyB_Array[n].Comms.Write.index := 83;
			IO_Link.EasyB.EasyB_Array[n].Comms.Write.subIndex := 0;
			IO_Link.EasyB.EasyB_Array[n].Comms.dataToWrite := n;
			IO_Link.EasyB.EasyB_Array[n].Comms.Write.pData := ADR(IO_Link.EasyB.EasyB_Array[n].Comms.dataToWrite);
			IO_Link.EasyB.EasyB_Array[n].Comms.Write.dataLen := 1;
			IO_Link.EasyB.EasyB_Array[n].Comms.Write.datatype := ioLinkTYPE_USINT;
			IO_Link.EasyB.EasyB_Array[n].Comms.Write();
			//Goto next state
			IF IO_Link.EasyB.EasyB_Array[n].Comms.Write.status <> ERR_FUB_BUSY THEN
				IO_Link.EasyB.EasyB_Array[n].Cmd.ClearCounter := FALSE;
			END_IF;
		ELSIF IO_Link.EasyB.EasyB_Array[n].Cmd.SetTripCurrent > 0 THEN
			//Specific function config
			IO_Link.EasyB.EasyB_Array[n].Comms.Write.index := 400 + n;
			IO_Link.EasyB.EasyB_Array[n].Comms.Write.subIndex := 0;
			IO_Link.EasyB.EasyB_Array[n].Comms.Write.pData := ADR(IO_Link.EasyB.EasyB_Array[n].Cmd.SetTripCurrent);
			IO_Link.EasyB.EasyB_Array[n].Comms.Write.dataLen := 1;
			IO_Link.EasyB.EasyB_Array[n].Comms.Write.datatype := ioLinkTYPE_USINT;
			IO_Link.EasyB.EasyB_Array[n].Comms.Write();
			//Goto next state
			IF IO_Link.EasyB.EasyB_Array[n].Comms.Write.status <> ERR_FUB_BUSY THEN
				IO_Link.EasyB.EasyB_Array[n].Cmd.SetTripCurrent := 0;
			END_IF;
		END_IF;
	END_FOR;
END_ACTION
```

#### _Contactron.st
```iecst
ACTION _Contactron:
	//----------------------------------------------
	//-----------------Contactron-------------------
	//----------------------------------------------

	//Write control word
	FOR n:=1 TO MAX_CONTACTRON DO
		IO_Link.Contactron[n].Comms.Read.CurrentActual := IO_Link.Contactron[n].Comms.Read.Data[0];
		IO_Link.Contactron[n].Comms.Read.DeviceType := IO_Link.Contactron[n].Comms.Read.Data[1];
		IO_Link.Contactron[n].Comms.Read.ThermalPercentOfMax := IO_Link.Contactron[n].Comms.Read.Data[2];
		IO_Link.Contactron[n].Comms.Read.CurrentPercentOfMax := IO_Link.Contactron[n].Comms.Read.Data[3];
		IO_Link.Contactron[n].Comms.Read.CurrentStatus := IO_Link.Contactron[n].Comms.Read.Data[4];
		IO_Link.Contactron[n].Comms.Read.Diagnostics := IO_Link.Contactron[n].Comms.Read.Data[5];

		//Read status
		IO_Link.Contactron[n].Status.Error := IO_Link.Contactron[n].Comms.Read.Diagnostics.0;
		IO_Link.Contactron[n].Status.STO_Active := NOT IO_Link.Contactron[n].Comms.Read.Diagnostics.3;
		IO_Link.Contactron[n].Status.Device_Ok := IO_Link.Contactron[n].Comms.Read.Diagnostics.5;
		IO_Link.Contactron[n].Status.Overload_Warning := IO_Link.Contactron[n].Comms.Read.Diagnostics.6;
		IO_Link.Contactron[n].Status.MainsFailure := ((IO_Link.Contactron[n].Comms.Read.CurrentStatus AND CONTACTRON_TRIP_STATUS) = CONTACTRON_MAINS_LOSS);
		IO_Link.Contactron[n].Status.PhaseLoss := ((IO_Link.Contactron[n].Comms.Read.CurrentStatus AND CONTACTRON_TRIP_STATUS) = CONTACTRON_PHASE_LOSS);
		IO_Link.Contactron[n].Status.Current := IO_Link.Contactron[n].Comms.Read.CurrentActual * 0.01;
		IO_Link.Contactron[n].Status.DeviceType := IO_Link.Contactron[n].Comms.Read.DeviceType;

		CASE IO_Link.Contactron[n].Cmd.Direction OF
			CONTACTRON_FORWARD:
				IO_Link.Contactron[n].Comms.Write.Control.0 := IO_Link.Contactron[n].Cmd.Run AND NOT IO_Link.Contactron[n].Status.Error;
				IO_Link.Contactron[n].Comms.Write.Control.7 := IO_Link.Contactron[n].Cmd.Run AND NOT IO_Link.Contactron[n].Status.Error;
				IO_Link.Contactron[n].Comms.Write.Control.1 := FALSE;
				IO_Link.Contactron[n].Comms.Write.Control.5 := FALSE;

			CONTACTRON_REVERSE:
				IO_Link.Contactron[n].Comms.Write.Control.0 := FALSE;
				IO_Link.Contactron[n].Comms.Write.Control.7 := FALSE;
				IO_Link.Contactron[n].Comms.Write.Control.1 := IO_Link.Contactron[n].Cmd.Run AND NOT IO_Link.Contactron[n].Status.Error;
				IO_Link.Contactron[n].Comms.Write.Control.5 := IO_Link.Contactron[n].Cmd.Run AND NOT IO_Link.Contactron[n].Status.Error;

			ELSE
				IO_Link.Contactron[n].Comms.Write.Control.0 := FALSE;
				IO_Link.Contactron[n].Comms.Write.Control.7 := FALSE;
				IO_Link.Contactron[n].Comms.Write.Control.1 := FALSE;
				IO_Link.Contactron[n].Comms.Write.Control.5 := FALSE;

		END_CASE;

		IO_Link.Contactron[n].Comms.Write.Control.2 := IO_Link.Contactron[n].Cmd.Reset_Manual;
		IO_Link.Contactron[n].Comms.Write.Control.3 := IO_Link.Contactron[n].Cmd.Reset_Automatic;
		IO_Link.Contactron[n].Comms.Write.Control.4 := FALSE; //NOT USED
		IO_Link.Contactron[n].Comms.Write.Control.6 := IO_Link.Contactron[n].Cmd.Stop;

		IF IO_Link.Contactron[n].Cmd.Current > 0 THEN //Write trip current level
			IO_Link.Contactron[n].Comms.Write.NominalCurrent := (IO_Link.Contactron[n].Cmd.Current OR CONTACTRON_WRITE_CURRENT);
		ELSE
			IO_Link.Contactron[n].Comms.Write.NominalCurrent := 0;
		END_IF;
		IF IO_Link.Contactron[n].Cmd.Current = (IO_Link.Contactron[n].Comms.Read.CurrentStatus AND CONTACTRON_CURRENT_STATUS) THEN
			IO_Link.Contactron[n].Cmd.Current := 0; //Reset trip current if cmd written
		END_IF;

	END_FOR;
END_ACTION
```

#### _status.st
```iecst
ACTION _status:
	CASE statusState OF
		0:
			offset := 1;
			FOR n:=1 TO MAX_CONTACTRON DO
				statusValue[n] := IO_Link.Contactron[n].Status.Current;
				offset := offset + 1;
			END_FOR;
			offset := MAX_CONTACTRON;
//			FOR n:=1 TO MAX_EASYB DO
//				statusValue[offset + n] := INT_TO_REAL(IO_Link.EasyB.EasyB_Array[n].Status.Current);
//				offset := offset + 1;
//			END_FOR;
			statusState := 1;
		1:
//			memset(ADR(IO_Link.httpRequest),0,SIZEOF(IO_Link.httpRequest));
//			ftoa(MAX_CONTACTRON,ADR(tempString));
//			strcat(ADR(IO_Link.httpRequest),ADR(tempString));
//			strcat(ADR(IO_Link.httpRequest),ADR(","));
//			ftoa(MAX_EASYB,ADR(tempString));
//			strcat(ADR(IO_Link.httpRequest),ADR(tempString));
//			strcat(ADR(IO_Link.httpRequest),ADR(","));
//			FOR n:=1 TO offset DO
//				ftoa(statusValue[n],ADR(tempString));
//				strcat(ADR(IO_Link.httpRequest),ADR(tempString));
//				strcat(ADR(IO_Link.httpRequest),ADR(","));
//			END_FOR;
//			statusState := 0;
//			IO_Link.Status := FALSE;
	END_CASE;

END_ACTION
```

#### backUpWrite.st
```iecst
ACTION _backUpWrite:
	IF (backUp.step = backUpExit) OR (backUp.step = backUpErrorRead) THEN
		backUp.step := backUpOpen;
	END_IF;
		CASE backUp.step OF
			backUpOpen:
				backUp.functions.fOpen.enable := TRUE;
				backUp.functions.fOpen.pDevice := ADR(backUp.fileDevice);
				backUp.functions.fOpen.pFile := ADR(backUp.filePath);
				backUp.functions.fOpen.mode := FILE_RW;
				backUp.functions.fOpen();
				backUp.ident := backUp.functions.fOpen.ident;
				backUp.status := backUp.functions.fOpen.status;
				IF (backUp.status = fiERR_FILE_NOT_FOUND) THEN
					backUp.step := backUpCreate; //File not found goto creat file step
				ELSIF (backUp.status = ERR_OK) THEN
					backUp.step := backUpWrite;	//File opened goto file write
				ELSIF (backUp.status = ERR_FUB_BUSY) THEN
					backUp.step := backUpOpen; //Function block still busy
				ELSE
					backUp.step := backUpErrorWrite; //Error goto error step
				END_IF;

			backUpCreate:
				backUp.functions.fCreate.enable := TRUE;
				backUp.functions.fCreate.pDevice := ADR(backUp.fileDevice);
				backUp.functions.fCreate.pFile := ADR(backUp.filePath);
				backUp.functions.fCreate();
				backUp.ident := backUp.functions.fCreate.ident;
				backUp.status := backUp.functions.fCreate.status;
				IF (backUp.status = ERR_OK) THEN
					backUp.step := backUpWrite;	//File created goto file write
				ELSIF (backUp.status = ERR_FUB_BUSY) THEN
					backUp.step := backUpCreate; //Function block still busy
				ELSE
					backUp.step := backUpErrorWrite; //Error goto error step
				END_IF;

			backUpWrite:
				backUp.functions.fWrite.enable := TRUE;
				backUp.functions.fWrite.ident := backUp.ident;
				backUp.functions.fWrite.offset := 0;
				backUp.functions.fWrite.pSrc := ADR(fuseSettingStructure);
				backUp.functions.fWrite.len := SIZEOF(fuseSettingStructure);
				backUp.functions.fWrite();
				backUp.status := backUp.functions.fWrite.status;
				IF (backUp.status = ERR_OK) THEN
					backUp.step := backUpClose; //Goto close file
				ELSIF (backUp.status = ERR_FUB_BUSY) THEN
					backUp.step := backUpWrite; //Function block still busy
				ELSE
					backUp.step := backUpErrorWrite; //Error goto error step
				END_IF;

			backUpClose:
				backUp.functions.fClose.enable := TRUE;
				backUp.functions.fClose.ident := backUp.ident;
				backUp.functions.fClose();
				backUp.status := backUp.functions.fClose.status;
				IF (backUp.status = ERR_OK) THEN
				//Exit case and action
					IO_Link.Save := FALSE;
					backUp.step := backUpExit;
				ELSIF (backUp.status = ERR_FUB_BUSY) THEN
					backUp.step := backUpClose; //Function block still busy
				ELSE
					backUp.step := backUpErrorWrite; //Error goto error step
				END_IF;

			backUpErrorWrite:
			//Error state
			IO_Link.Save := FALSE;
	END_CASE;
END_ACTION
```

#### backUpRead.st
```iecst
ACTION _backUpRead:
	IF (backUp.step = backUpExit) THEN
		backUp.step := backUpOpen;
	END_IF;
	CASE backUp.step OF
			backUpOpen:
				backUp.functions.fOpen.enable := TRUE;
				backUp.functions.fOpen.pDevice := ADR(backUp.fileDevice);
				backUp.functions.fOpen.pFile := ADR(backUp.filePath);
				backUp.functions.fOpen.mode := FILE_RW;
				backUp.functions.fOpen();
				backUp.status := backUp.functions.fOpen.status;
				IF (backUp.status = fiERR_FILE_NOT_FOUND) THEN
					backUp.step := backUpErrorRead; //Error goto error step
				ELSIF (backUp.status = ERR_OK) THEN
					backUp.step := backUpRead;	//File opened goto read write
					backUp.ident := backUp.functions.fOpen.ident;
				ELSIF (backUp.status = ERR_FUB_BUSY) THEN
					backUp.step := backUpOpen; //Function block still busy
				ELSE
					backUp.step := backUpErrorRead; //Error goto error step
				END_IF;

			backUpRead:
				backUp.functions.fRead.enable := TRUE;
				backUp.functions.fRead.ident := backUp.ident;
				backUp.functions.fRead.offset := 0;
				backUp.functions.fRead.pDest := ADR(fuseSettingStructure);
				backUp.functions.fRead.len := SIZEOF(fuseSettingStructure);
				backUp.functions.fRead();
				backUp.status := backUp.functions.fRead.status;
				IF (backUp.status = fiERR_FILE_NOT_FOUND) THEN
					backUp.step := backUpExit; //File not found goto exit loop
				ELSIF (backUp.status = ERR_OK) THEN
					backUp.step := backUpClose;	//goto close file
				ELSIF (backUp.status = ERR_FUB_BUSY) THEN
					backUp.step := backUpRead; //Function block still busy
				ELSE
					backUp.step := backUpErrorRead; //Error goto error step
				END_IF;

			backUpClose:
				backUp.functions.fClose.enable := TRUE;
				backUp.functions.fClose.ident := backUp.ident;
				backUp.functions.fClose();
				backUp.status := backUp.functions.fClose.status;
				IF (backUp.status = ERR_OK) THEN
					//Exit case and action
					IO_Link.Load := FALSE;
					backUp.step := backUpExit;
				ELSIF (backUp.status = ERR_FUB_BUSY) THEN
					backUp.step := backUpClose; //Function block still busy
				ELSE
					backUp.step := backUpErrorRead; //Error goto error step
				END_IF;

			backUpErrorRead:
				IO_Link.Load := FALSE;
				//Error state
		END_CASE;
END_ACTION
```

#### encodeData.st
```iecst
ACTION _encodeData:
	//Clear string memory
	memset(ADR(IO_Link.httpRequest),0,SIZEOF(IO_Link.httpRequest));
	//Add length to start of string
	ftoa(MAX_CONTACTRON,ADR(tempString));
	strcat(ADR(IO_Link.httpRequest),ADR(tempString));
	strcat(ADR(IO_Link.httpRequest),ADR(","));
	ftoa(MAX_EASYB,ADR(tempString));
	strcat(ADR(IO_Link.httpRequest),ADR(tempString));
	strcat(ADR(IO_Link.httpRequest),ADR(","));
	//Encode data
	FOR n:=1 TO MAX_CONTACTRON DO
		ftoa(fuseSettingStructure.Contactron[n],ADR(tempString));
		strcat(ADR(IO_Link.httpRequest),ADR(tempString));
		strcat(ADR(IO_Link.httpRequest),ADR(","));
	END_FOR;
	FOR n:=1 TO MAX_EASYB DO
		ftoa(fuseSettingStructure.EasyB[n],ADR(tempString));
		strcat(ADR(IO_Link.httpRequest),ADR(tempString));
		strcat(ADR(IO_Link.httpRequest),ADR(","));
	END_FOR;

	FOR n:=1 TO MAX_EASYB DO
		IO_Link.EasyB.EasyB_Array[n].Cmd.SetTripCurrent := fuseSettingStructure.EasyB[n];
	END_FOR;
	FOR n:=1 TO MAX_CONTACTRON DO
		IO_Link.Contactron[n].Cmd.Current := fuseSettingStructure.Contactron[n];
	END_FOR;
END_ACTION
```

#### decodeData.st
```iecst
ACTION _decodeData:

	state := CONTACTRON;
	count := 1;
	memset(ADR(tempString),0,SIZEOF(tempString));

	FOR loop:=0 TO SIZEOF(IO_Link.httpResponse) - 1 DO
		IF IO_Link.httpResponse[loop] = 0 THEN //Null
			EXIT;
		ELSIF IO_Link.httpResponse[loop] = 44 THEN //Comma
			CASE state OF
				CONTACTRON:
					fuseSettingStructure.Contactron[count] := DINT_TO_USINT(atoi(ADR(tempString)));
					count := count + 1;
					IF count > MAX_CONTACTRON THEN state := EASYB; count := 1; END_IF;
				EASYB:
					CASE DINT_TO_USINT(atoi(ADR(tempString))) OF
						TRIP_CURRENT_DEFAULT:
							fuseSettingStructure.EasyB[count] := TRIP_CURRENT_DEFAULT;
						TRIP_CURRENT_500mA:
							fuseSettingStructure.EasyB[count] := TRIP_CURRENT_500mA;
						TRIP_CURRENT_1A:
							fuseSettingStructure.EasyB[count] := TRIP_CURRENT_1A;
						TRIP_CURRENT_2A:
							fuseSettingStructure.EasyB[count] := TRIP_CURRENT_2A;
						TRIP_CURRENT_3A:
							fuseSettingStructure.EasyB[count] := TRIP_CURRENT_3A;
						TRIP_CURRENT_4A:
							fuseSettingStructure.EasyB[count] := TRIP_CURRENT_4A;
						TRIP_CURRENT_5A:
							fuseSettingStructure.EasyB[count] := TRIP_CURRENT_5A;
						TRIP_CURRENT_6A:
							fuseSettingStructure.EasyB[count] := TRIP_CURRENT_6A;
						TRIP_CURRENT_8A:
							fuseSettingStructure.EasyB[count] := TRIP_CURRENT_8A;
						TRIP_CURRENT_10A:
							fuseSettingStructure.EasyB[count] := TRIP_CURRENT_10A;
					END_CASE;
					count := count + 1;
			END_CASE;
			memset(ADR(tempString),0,SIZEOF(tempString));
		ELSE
			itoa(IO_Link.httpResponse[loop]-48, ADR(tempString2));
			tempString := CONCAT(tempString, tempString2);
		END_IF;
	END_FOR;

END_ACTION
```

### Modules.var
```iecst
VAR
	BusCouplerDiag : ARRAY[0..MAX_BUS_COUPLERS] OF BusCouplerDiag_typ;
END_VAR
VAR CONSTANT
	MAX_BUS_COUPLERS : UINT := 256;
END_VAR
```

### Modules.typ
```iecst
TYPE
	BusCouplerDiag_typ : 	STRUCT
		ModuleLostWhilstOperational : DINT;
		StationAtBusEnd : USINT;
		StationPastInFrameError : USINT;
		StationPastOutFrameError : USINT;
	END_STRUCT;
END_TYPE
```

### Program Logical/Standard/ModuleLogger/moduleWatch (IEC)

#### Variables.var
```iecst
VAR
	mpAuditTrail : MpAuditTrail;
	test : USINT;
	n : USINT;
	export : BOOL;
	clearBuffer : BOOL;
	busCouplerVisu : REFERENCE TO BusCouplerDiag_typ;
	index : USINT;
	timebase : UINT;
END_VAR
```

#### Main.st
```iecst
PROGRAM _INIT
BusCouplerDiag[31]; // ADD Reference to structure so AS builds correctl

mpAuditTrail.MpLink := ADR(gAuditTrail);
mpAuditTrail.DeviceName := ADR('user');
mpAuditTrail.Enable := 1;
test := 0;
timebase := 600;// 10mins.

END_PROGRAM

PROGRAM _CYCLIC

	IF (index > 0) AND (index <= MAX_BUS_COUPLERS) THEN
		busCouplerVisu ACCESS ADR(BusCouplerDiag[index]);
	ELSE
		busCouplerVisu ACCESS ADR(BusCouplerDiag[0]);
	END_IF;

	IF test > 0 THEN
		IF test < 16#FF THEN
			test := test + 1;
		ELSE
			test := 1;
		END_IF;
		n := 13;
		//FOR n := 31 TO 44 DO
		BusCouplerDiag[n].ModuleLostWhilstOperational := test;
		BusCouplerDiag[n].StationAtBusEnd := test;
		BusCouplerDiag[n].StationPastInFrameError := test;
		BusCouplerDiag[n].StationPastOutFrameError := test;
		//END_FOR;
	END_IF;

	mpAuditTrail.Export := export;
	mpAuditTrail();

	IF export AND mpAuditTrail.CommandDone THEN
		export := 0;
	END_IF;

	IF clearBuffer THEN
		MpAuditClearBuffer(gAuditTrail);
		clearBuffer := 0;
	END_IF;

	//New functions found in the B&R library to report IO execptions.
	//Can only be used in the excpetion task class.
	//IO_info_0(enable := 1);
	//IX_info_0(enable := 1);
	//
	//IO_info_0.enable := 1;
	//IO_info_0();

END_PROGRAM
PROGRAM _EXIT
	mpAuditTrail.Enable := 0; // Release the mappLink
	mpAuditTrail();
END_PROGRAM
```

### Package Logical/Standard/Settings - Looks after all PLC settings for drivers.

### Settings.var
```iecst
VAR RETAIN
	gSettings : {REDUND_UNREPLICABLE} settings_typ := (0);
END_VAR
```

### Settings.typ
```iecst
TYPE
	settings_typ : 	STRUCT
		Camera : ARRAY[0..MAX_CAMERAS]OF Camera_Settings_typ;
		Drive : ARRAY[0..MAX_DRIVES]OF ABB_Settings_typ;
		Rail : ARRAY[0..MAX_RAILS]OF Rail_Permenant_typ;
		Fuse : ARRAY[0..MAX_FUSE_BANKS]OF FuseSetting_typ;
		Contactron : ARRAY[0..MAX_CONTACTRON]OF contactron_setting_typ;
	END_STRUCT;
	Rail_Permenant_typ : 	STRUCT
		State : INT;
		Count : INT;
	END_STRUCT;
END_TYPE
```

### Program Logical/Standard/Settings/Permenant (IEC, version 2.00.1) - *Store/Restore memory

#### Main.st - Init, cyclic, exit code
```iecst
PROGRAM _INIT
//Set all the rail states to perm.

FOR n := 1 TO MAX_RAILS DO
  //build the var_name;

  pSettings.Rail_Counter[n] := ADR(gSettings.Rail[n].Count);
  pSettings.Rail_State[n] := ADR(gSettings.Rail[n].State);

  itoa(n,ADR(index_string));
  //r109.state
  var_name := 'r';
  brsstrcat(ADR(var_name),ADR(index_string));
  brsstrcat(ADR(var_name),ADR('.state'));
  // Get the Pointer address.
  IF (PV_xgetadr(ADR(var_name),ADR(pVar),ADR(sVar)) = 0) THEN
    p.Rail_State[n] := pVar;
    brsmemcpy(p.Rail_State[n],pSettings.Rail_State[n],2);
  ELSE
    p.Rail_State[n] := 0;
  END_IF;

  var_name := 'r';
  brsstrcat(ADR(var_name),ADR(index_string));
  brsstrcat(ADR(var_name),ADR('.counter'));
  IF (PV_xgetadr(ADR(var_name),ADR(pVar),ADR(sVar)) = 0) THEN
    p.Rail_Counter[n] := pVar;
    brsmemcpy(p.Rail_Counter[n],pSettings.Rail_Counter[n],2);
  ELSE
    p.Rail_Counter[n] := 0;
  END_IF;
END_FOR;

END_PROGRAM

PROGRAM _CYCLIC
(*******************************
Update belt speeds.
*******************************)
// Set the values from eVue.

beltSpeed[1] := Get_HigherByte(conveyor_module_1_value_1);
beltSpeed[2] := Get_LowerByte(conveyor_module_1_value_1);
beltSpeed[3] := Get_HigherByte(conveyor_module_1_value_2);
beltSpeed[4] := Get_LowerByte(conveyor_module_1_value_2);
//beltSpeed[5] := Get_HigherByte(conveyor_module_1_value_3);
//beltSpeed[6] := Get_LowerByte(conveyor_module_1_value_3);
//
FOR n := 1 TO MAX_DRIVES DO
  IF (beltSpeed[n] > 0) AND (beltSpeed[n] <> gSettings.Drive[n].TargetVelocity) THEN
    gSettings.Drive[n].TargetVelocity := beltSpeed[n];
  ELSIF (gSettings.Drive[n].TargetVelocity = 0) THEN
    gSettings.Drive[n].TargetVelocity := ABB_MAX_VELOCITY;
  END_IF;
END_FOR;

FOR n := 1 TO MAX_RAILS DO
  IF (p.Rail_Counter[n] > 0) AND (pSettings.Rail_Counter[n] > 0) THEN
    brsmemcpy(pSettings.Rail_Counter[n],p.Rail_Counter[n],2);
  END_IF;
  IF (p.Rail_State[n] > 0) AND (pSettings.Rail_State[n] > 0) THEN
    brsmemcpy(pSettings.Rail_State[n],p.Rail_State[n],2);
  END_IF;

END_FOR;

END_PROGRAM
```

#### Types.typ - Local data types
```iecst
TYPE
	Pointer_typ : 	STRUCT
		Rail_Counter : ARRAY[0..MAX_RAILS]OF UDINT;
		Rail_State : ARRAY[0..MAX_RAILS]OF UDINT;
	END_STRUCT;
END_TYPE
```

#### Variables.var - Local variables
```iecst
VAR
	beltSpeed : ARRAY[0..MAX_DRIVES] OF INT;
	n : UINT;
	var_name : STRING[50];
	var_value : UDINT;
	index_string : STRING[10];
	init : BOOL;
	pSettings : Pointer_typ;
	p : Pointer_typ;
	sVar : UDINT;
	pVar : UDINT;
END_VAR
```

### Program Logical/Standard/ToDO/light_towers (IEC)

#### Variables.var
```iecst
VAR
	AlarmOutput : ARRAY[0..MAX_SYSTEMS] OF BOOL;
	safeZone : REFERENCE TO SafeZoneType;
	tmrAlmOutput : ARRAY[0..MAX_SYSTEMS] OF TON;
	n : USINT;
	myZone : ARRAY[0..MAX_SYSTEMS] OF USINT;
END_VAR
VAR CONSTANT
	MAX_SYSTEMS : USINT := 2;
END_VAR
```

#### Main.st
```iecst
PROGRAM _INIT
  myZone[1] := 1;
  myZone[2] := 11;
END_PROGRAM

PROGRAM _CYCLIC
  // Soiled Tower
  AlarmOutput[1] := system_alarm_2 OR soiled_validation_alarm OR halted;
  AlarmOutput[2] := system_alarm_1 OR clean_validation_alarm OR halted;

  FOR n := 1 TO MAX_SYSTEMS DO
    safeZone ACCESS ADR(SafetyZone[myZone[n]]);

    tmrAlmOutput[n].IN := AlarmOutput[n];
    tmrAlmOutput[n].PT := T#5s;
    tmrAlmOutput[n]();

    safeZone.TowerLight.TL_DO_Red 		:= FALSE;
    safeZone.TowerLight.TL_DO_Yellow	:= FALSE;
    safeZone.TowerLight.TL_DO_Green	:= FALSE;
    IF safeZone.HaltSys AND NOT safeZone.ResetReady THEN	//Emergency stop blink red. (State 1)
      safeZone.TowerLight.TL_DO_Red 		:= Std.Clock1s ;
    ELSIF safeZone.HaltSys THEN // Estop waiting for reset  (State 2)
      safeZone.TowerLight.TL_DO_Yellow		:= Std.Clock1s;
    ELSIF AlarmOutput[n] THEN //State 10 -- Show Warning Not Fault when alarm is on as other parts might still be running
      safeZone.TowerLight.TL_DO_Yellow 	:= TRUE;
      safeZone.TowerLight.TL_DO_Green	 := TRUE;
    ELSE //Machine Running (State 6)
      safeZone.TowerLight.TL_DO_Green	 := TRUE;
    END_IF;
    safeZone.TowerLight.TL_DO_Sounder := (AlarmOutput[n] AND NOT tmrAlmOutput[n].Q);
  END_FOR;

END_PROGRAM
```

### Library Logical/Standard/FileMgr (IEC)
Depends on: FileIO, DataObj, AsHttp

#### Types.typ - Exported data types
```iecst
TYPE
	fileToDatObj_state :
		(
		Fi_To_Do_INIT,
		Fi_To_Do_FILE_OPEN,
		Fi_To_Do_FILE_READ,
		Fi_To_Do_FILE_CLOSE,
		Fi_To_Do_DObj_GET_INFO,
		Fi_To_Do_DObj_DELETE,
		Fi_To_Do_DObj_CREATE,
		Fi_To_Do_ERROR,
		Fi_To_Do_DObj_WRITE
		);
	fileToMem_state :
		(
		Fi_To_Mem_INIT,
		Fi_To_Mem_FILE_OPEN,
		Fi_To_Mem_FILE_READ,
		Fi_To_Mem_FILE_CLOSE,
		Fi_To_Mem_ERROR
		);
	fileCopyFromDev_state :
		(
		FiCopyDev_INIT,
		FiCopyDev_DEVLINK,
		FiCopyDev_COPY,
		FiCopyDev_UNLINK,
		FiCopyDev_ERROR
		);

END_TYPE
```

#### Constants.var - Exported constants
```iecst
(*FILE READ WRITE INTERNAL STATES*)
VAR CONSTANT
	FILE_STATE_OPEN : UINT := 1;
	FILE_STATE_CREATE : UINT := 10;
	FILE_STATE_WRITE : UINT := 20;
	FILE_STATE_READ : UINT := 30;
	FILE_STATE_CLOSE : UINT := 40;
	FILE_STATE_ERROR : UINT := 99;
END_VAR
(*FILE READ WRITE INPUT MODES*)
VAR CONSTANT
	FILE_SAVE : UINT := 0;
	FILE_READ : UINT := 1;
END_VAR
```

#### FileMgr.fun - Exported functions and function blocks
```iecst
FUNCTION_BLOCK fileReadWrite (**Read or Write to file*) (*$GROUP=User,$CAT=User,$GROUPICON=User.png,$CATICON=User.png*)
	VAR_INPUT
		enable : BOOL;
		pFileDevice : UDINT;
		pFileName : UDINT;
		mode : UINT;
		pData : UDINT; (*point to data to read or write to*)
		sizeData : UDINT; (*size of data to read or write to*)
		Offset : UDINT; (*offset of data to be read or written*)
		appendToFile : BOOL;
	END_VAR
	VAR_OUTPUT
		status : UINT;
	END_VAR
	VAR
		fileState : UINT;
		fileOpen : FileOpen;
		fileCreate : FileCreate;
		fileClose : FileClose;
		error : UINT;
		fileWrite : FileWrite;
		ident : UDINT;
		fileRead : FileRead;
	END_VAR
END_FUNCTION_BLOCK

FUNCTION_BLOCK fileToDatObj (**read from a file into a data object. The data object will be deleted and created the same size as file*) (*$GROUP=User,$CAT=User,$GROUPICON=User.png,$CATICON=User.png*)
	VAR_INPUT
		enable : BOOL; (** Enable*)
		pFileDevice : UDINT; (*pointer to file device*)
		pFileName : UDINT; (*pointer to the file name*)
		pDoName : UDINT; (*pointer to the name of the dataObject to be written to*)
		MemType : USINT;
	END_VAR
	VAR_OUTPUT
		status : UINT;
		do_Ident : UDINT; (*pointer to the ident to the data Object*)
		pDatObjMem : UDINT; (*Pointer to the memory area of the data object written to*)
		fiSize : UDINT;
	END_VAR
	VAR
		fileOpen : FileOpen;
		error : UINT;
		fileRead : FileRead;
		fileClose : FileClose;
		fileState : fileToDatObj_state;
		fi_ident : UDINT;
		do_GetInfo : DatObjInfo;
		do_Delete : DatObjDelete;
		do_Create : DatObjCreate;
		do_Write : DatObjWrite;
	END_VAR
END_FUNCTION_BLOCK

FUNCTION_BLOCK fileToMem (**OpenFileInto memory*) (*$GROUP=User,$CAT=User,$GROUPICON=User.png,$CATICON=User.png*)
	VAR_INPUT
		enable : BOOL; (** Enable*)
		pFileDevice : UDINT; (*pointer to file device*)
		pFileName : UDINT; (*pointer to the file name*)
		pTempMem : UDINT; (**point to the memory area created by TMP_alloc*)
		sizeTempMem : UDINT; (**Size of the temporary memory allocated by TMP_alloc*)
	END_VAR
	VAR_OUTPUT
		status : UINT;
		fiSize : UDINT;
	END_VAR
	VAR
		fileOpen : FileOpen;
		error : UINT;
		fileRead : FileRead;
		fileClose : FileClose;
		fileState : fileToMem_state;
		fi_ident : UDINT;
	END_VAR
END_FUNCTION_BLOCK

FUNCTION_BLOCK FileCopyFromDev (**Copy file from devlink link file device*) (*$GROUP=User,$CAT=User,$GROUPICON=User.png,$CATICON=User.png*)
	VAR_INPUT
		enable : BOOL;
		pFileDevice : UDINT;
		pDevLinkParameter : UDINT;
		pFileName : UDINT;
		pDest : UDINT;
		pDestDev : UDINT;
	END_VAR
	VAR_OUTPUT
		status : UINT;
	END_VAR
	VAR
		fileState : fileCopyFromDev_state;
		error : UINT;
		devLink : DevLink;
		fileCopy : FileCopy;
		devUnlink : DevUnlink;
		devHandle : UDINT;
	END_VAR
END_FUNCTION_BLOCK
```

#### fileToDatObj.st - *Gives Check sum errors -- Use fileToMem
```iecst
(* *read from a file into a data object. *)
FUNCTION_BLOCK fileToDatObj

	IF enable THEN
		CASE fileState OF
			Fi_To_Do_INIT:
				pDatObjMem := 0;
				fileState := Fi_To_Do_FILE_OPEN;
				status := ERR_FUB_BUSY;
				error := 0;

			Fi_To_Do_FILE_OPEN:
				fileOpen.enable := 1;
				fileOpen.pDevice := pFileDevice;
				fileOpen.pFile := pFileName;
				fileOpen.mode := fiREAD_WRITE;
				fileOpen();
				IF fileOpen.status = ERR_OK THEN
					fi_ident := fileOpen.ident;
					fiSize := fileOpen.filelen;
					fileState := Fi_To_Do_DObj_GET_INFO;
				ELSIF fileOpen.status = fiERR_FILE_NOT_FOUND THEN
					fileState := Fi_To_Do_ERROR;
					status := fileOpen.status;
				ELSIF fileOpen.status <> ERR_FUB_BUSY THEN
					fileState := Fi_To_Do_ERROR;
					status := fileOpen.status;
				END_IF;

			Fi_To_Do_DObj_GET_INFO:
				do_GetInfo.enable := 1;
				do_GetInfo.pName := pDoName;
				do_GetInfo();
				IF do_GetInfo.status = ERR_OK THEN
					do_Ident := do_GetInfo.ident;
					fileState := Fi_To_Do_DObj_DELETE;
				ELSIF do_GetInfo.status = doERR_MODULNOTFOUND THEN
					fileState := Fi_To_Do_DObj_CREATE;
				ELSIF do_GetInfo.status <> ERR_FUB_BUSY THEN
					fileState := Fi_To_Do_FILE_CLOSE;
					error := do_GetInfo.status;
				END_IF;

			Fi_To_Do_DObj_DELETE:
				do_Delete.enable := 1;
				do_Delete.ident := do_Ident;
				do_Delete();
				IF do_Delete.status = ERR_OK THEN
					fileState := Fi_To_Do_DObj_CREATE;
				ELSIF do_Delete.status <> ERR_FUB_BUSY THEN
					fileState := Fi_To_Do_FILE_CLOSE;
					error := do_Delete.status;
				END_IF;

			Fi_To_Do_DObj_CREATE:
				do_Create.enable 	:= 1;
				do_Create.pName 	:= pDoName;
				do_Create.Option 	:= doNO_CS; // No checksum if do not call the DatObjWrite FUB>
				do_Create.pCpyData 	:= 0;
				do_Create.MemType	:= MemType;// doUSRROM;
				do_Create.len		:= fiSize;
				do_Create();
				IF (do_Create.status = ERR_OK) OR (do_Create.status = doERR_CHECKSUM_WARNING) THEN
					do_Ident := do_Create.ident;
					pDatObjMem	:= do_Create.pDatObjMem;
					fileState := Fi_To_Do_FILE_READ;
				ELSIF do_Create.status <> ERR_FUB_BUSY THEN
					error := do_Create.status;
					fileState := Fi_To_Do_FILE_CLOSE;
				END_IF;

			Fi_To_Do_FILE_READ:
				fileRead.enable := 1;
				fileRead.ident := fi_ident;
				fileRead.pDest := pDatObjMem;
				fileRead.len := fiSize;
				fileRead.offset := 0;
				fileRead();
				IF fileRead.status = ERR_OK THEN
					fileState := Fi_To_Do_FILE_CLOSE;
				ELSIF fileRead.status <> ERR_FUB_BUSY THEN
					error := fileRead.status;
					fileState := Fi_To_Do_FILE_CLOSE;
				END_IF;

			Fi_To_Do_DObj_WRITE:
				do_Write.enable := 1;
				do_Write.ident := do_Ident;
				do_Write.Offset := 0;
				do_Write.len := fiSize;
				do_Write.pSource := pDatObjMem;
				do_Write();
				IF do_Write.status = ERR_OK	 THEN
					fileState := Fi_To_Do_FILE_CLOSE;
				ELSIF do_Write.status <> ERR_FUB_BUSY THEN
					error := fileRead.status;
					fileState := Fi_To_Do_FILE_CLOSE;
				END_IF;

			Fi_To_Do_FILE_CLOSE:
				fileClose.enable := 1;
				fileClose.ident := fi_ident;
				fileClose();
				IF fileClose.status = ERR_OK THEN
					IF (error > 0) THEN
						status := error;
						fileState := Fi_To_Do_ERROR;
					ELSE
						status := ERR_OK;
						fileState := Fi_To_Do_INIT; //Reset FUB
					END_IF;
				ELSIF fileClose.status <> ERR_FUB_BUSY THEN
					fileState := Fi_To_Do_ERROR;
					status := fileClose.status;
				END_IF;

			Fi_To_Do_ERROR://Error!!
				fileState:= Fi_To_Do_INIT;

		END_CASE;
	ELSE
		error := 0;
		fileState := Fi_To_Do_INIT;
		status := ERR_FUB_ENABLE_FALSE;
	END_IF;

END_FUNCTION_BLOCK
```

#### fileReadWrite.st
```iecst
(* *Read or write to file device *)
FUNCTION_BLOCK fileReadWrite

	IF enable THEN
		CASE fileState OF
			0:
				IF mode	= FILE_SAVE THEN
					fileState := FILE_STATE_OPEN;
					status := ERR_FUB_BUSY;
				ELSIF mode = FILE_READ THEN
					fileState := FILE_STATE_OPEN;
					status := ERR_FUB_BUSY;
				ELSE
					fileState := FILE_STATE_ERROR;
					status := 99;//Incorrect config
				END_IF;

			FILE_STATE_OPEN:
				fileOpen.enable := 1;
				fileOpen.pDevice := pFileDevice; //MEMCARD
				fileOpen.pFile := pFileName;
				fileOpen.mode := fiREAD_WRITE;
				fileOpen();
				IF fileOpen.status = ERR_OK THEN

					ident := fileOpen.ident;
					IF mode = FILE_SAVE THEN
						fileState := FILE_STATE_WRITE;
						IF appendToFile THEN Offset := fileOpen.filelen; END_IF;
					ELSIF mode = FILE_READ THEN
						fileState := FILE_STATE_READ;
					END_IF;
				ELSIF fileOpen.status = fiERR_FILE_NOT_FOUND THEN
					IF mode = FILE_SAVE THEN
						fileState := FILE_STATE_CREATE;
					ELSE
						fileState := FILE_STATE_ERROR;
						status := fileOpen.status;
					END_IF;
				ELSIF fileOpen.status <> ERR_FUB_BUSY THEN
					fileState := FILE_STATE_ERROR;
					status := fileOpen.status;
				END_IF;

			FILE_STATE_CREATE:
				fileCreate.enable := 1;
				fileCreate.pDevice := pFileDevice;
				fileCreate.pFile := pFileName;
				fileCreate();
				IF fileCreate.status = ERR_OK THEN
					fileState := FILE_STATE_WRITE;
					ident := fileCreate.ident;
				ELSIF fileCreate.status <> ERR_FUB_BUSY THEN
					fileState := FILE_STATE_ERROR;
					status := fileCreate.status;
				END_IF;

			FILE_STATE_WRITE:
				fileWrite.enable := 1;
				fileWrite.ident := ident;
				fileWrite.pSrc := pData;
				fileWrite.len := sizeData;
				fileWrite.offset := Offset;
				fileWrite();
				IF fileWrite.status = ERR_OK THEN
					fileState := FILE_STATE_CLOSE;
				ELSIF fileWrite.status <> ERR_FUB_BUSY THEN
					error := fileWrite.status;
					fileState := FILE_STATE_CLOSE;
				END_IF;

			FILE_STATE_READ:
				fileRead.enable := 1;
				fileRead.ident := ident;
				fileRead.pDest := pData;
				fileRead.len := sizeData;
				fileRead.offset := Offset;
				fileRead();
				IF fileRead.status = ERR_OK THEN
					fileState := FILE_STATE_CLOSE;
				ELSIF fileRead.status <> ERR_FUB_BUSY THEN
					error := fileRead.status;
					fileState := FILE_STATE_CLOSE;
				END_IF;

			FILE_STATE_CLOSE:
				fileClose.enable := 1;
				fileClose.ident := ident;
				fileClose();
				IF fileClose.status = ERR_OK THEN
					IF (error > 0) THEN
						status := error;
						fileState := FILE_STATE_ERROR;
					ELSE
						status := ERR_OK;
						fileState := 0; //Reset FUB
					END_IF;
				ELSIF fileClose.status <> ERR_FUB_BUSY THEN
					fileState := FILE_STATE_ERROR;
					status := fileClose.status;
				END_IF;

			FILE_STATE_ERROR://Error!!
				fileState:= 0;

		END_CASE;
	ELSE
		error := 0;
		fileState := 0;
		status := ERR_FUB_ENABLE_FALSE;
	END_IF;

END_FUNCTION_BLOCK
```

#### fileToMem.st
```iecst
(* *Opens File Into memory area*)
FUNCTION_BLOCK fileToMem
	IF enable THEN
		CASE fileState OF
			Fi_To_Mem_INIT:
				fileState := Fi_To_Mem_FILE_OPEN;
				status := ERR_FUB_BUSY;
				error := 0;

			Fi_To_Mem_FILE_OPEN:
				fileOpen.enable := 1;
				fileOpen.pDevice := pFileDevice;
				fileOpen.pFile := pFileName;
				fileOpen.mode := fiREAD_ONLY;
				fileOpen();
				IF fileOpen.status = ERR_OK THEN
					fi_ident := fileOpen.ident;
					fiSize := fileOpen.filelen;
					IF fiSize <= sizeTempMem THEN
						fileState := Fi_To_Mem_FILE_READ;
					ELSE
						error := fiERR_NOT_ENOUGH_FREEMEM;
						fileState := Fi_To_Mem_FILE_CLOSE;
					END_IF;
				ELSIF fileOpen.status = fiERR_FILE_NOT_FOUND THEN
					fileState := Fi_To_Mem_ERROR;
					status := fileOpen.status;
				ELSIF fileOpen.status <> ERR_FUB_BUSY THEN
					fileState := Fi_To_Mem_ERROR;
					status := fileOpen.status;
				END_IF;

			Fi_To_Mem_FILE_READ:
				fileRead.enable := 1;
				fileRead.ident := fi_ident;
				fileRead.pDest := pTempMem;
				fileRead.len := fiSize;
				fileRead.offset := 0;
				fileRead();
				IF fileRead.status = ERR_OK THEN
					fileState := Fi_To_Mem_FILE_CLOSE;
				ELSIF fileRead.status <> ERR_FUB_BUSY THEN
					error := fileRead.status;
					fileState := Fi_To_Mem_FILE_CLOSE;
				END_IF;

			Fi_To_Mem_FILE_CLOSE:
				fileClose.enable := 1;
				fileClose.ident := fi_ident;
				fileClose();
				IF fileClose.status = ERR_OK THEN
					IF (error > 0) THEN
						status := error;
						fileState := Fi_To_Mem_ERROR;
					ELSE
						status := ERR_OK;
						fileState := Fi_To_Mem_INIT; //Reset FUB
					END_IF;
				ELSIF fileClose.status <> ERR_FUB_BUSY THEN
					fileState := Fi_To_Mem_ERROR;
					status := fileClose.status;
				END_IF;

			Fi_To_Mem_ERROR://Error!!
				fileState:= Fi_To_Mem_INIT;

		END_CASE;
	ELSE
		error := 0;
		fileState := Fi_To_Mem_INIT;
		status := ERR_FUB_ENABLE_FALSE;
	END_IF;

END_FUNCTION_BLOCK
```

#### FileCopyFromDev.st
```iecst
(* *Copy file from devlink link file device *)
FUNCTION_BLOCK FileCopyFromDev
	status := ERR_FUB_BUSY;
	IF enable THEN
		CASE fileState OF
			FiCopyDev_INIT:
				fileState := FiCopyDev_DEVLINK;
				status := ERR_FUB_BUSY;
				error := 0;

			FiCopyDev_DEVLINK:
				devLink.enable := 1;
				devLink.pDevice := pFileDevice;
				devLink.pParam := pDevLinkParameter;
				devLink();
				IF (devLink.status = ERR_OK) OR (devLink.status = fiERR_DEVICE_ALREADY_EXIST) THEN
					fileState := FiCopyDev_COPY;
					devHandle := devLink.handle; // Handle is not returned when fiERR_DEVICE_ALREADY_EXIST
				ELSIF devLink.status = fiERR_SYSTEM THEN
					status := FileIoGetSysError();
					fileState := FiCopyDev_ERROR;
				END_IF;

			FiCopyDev_COPY:
				fileCopy.enable := 1;
				fileCopy.pSrc := pFileName;
				fileCopy.pSrcDev := pFileDevice;
				fileCopy.pDest := pDest;
				fileCopy.pDestDev := pDestDev;
				fileCopy.option := fiOVERWRITE;
				fileCopy();
				IF fileCopy.status = ERR_OK THEN
					fileState := FiCopyDev_UNLINK;
				ELSIF fileCopy.status <> ERR_FUB_BUSY THEN
					error := fileCopy.status;
					fileState := FiCopyDev_UNLINK;
				END_IF;

			FiCopyDev_UNLINK:
				devUnlink.enable := (devHandle > 0);
				devUnlink.handle := devHandle;
				devUnlink();
				IF (devUnlink.status = ERR_OK) OR (devHandle = 0) THEN
					IF error = 0 THEN
						status := ERR_OK;
						fileState := FiCopyDev_INIT;
					ELSE
						fileState := FiCopyDev_ERROR;
					END_IF;
				ELSIF (devUnlink.status <> ERR_FUB_BUSY) THEN
					error := devUnlink.status;
					fileState := FiCopyDev_ERROR;
				END_IF;

			FiCopyDev_ERROR://Error!!
				status := error;
				error := 0;
				fileState:= FiCopyDev_INIT;

		END_CASE;
	ELSE
		error := 0;
		fileState := FiCopyDev_INIT;
		status := ERR_FUB_ENABLE_FALSE;
	END_IF;
END_FUNCTION_BLOCK
```

### Package Logical/Standard/Kanlink/Supertrack_Kanlink_Constants - *Kanlink constants

### Supertrack_Constants.var - Global variables
```iecst
(********************************************************************
 * COPYRIGHT -- HP
 ********************************************************************
 * Package: Supertrack_Constants
 * File: Supertrack_Constants.var
 * Author: treamsbottom
 * Created: January 28, 2013
 ********************************************************************
 * Variables of package Supertrack_Constants
 ********************************************************************)
VAR CONSTANT
	BatchTyp_UDINT : USINT := 0;
	BatchTyp_16Byte : USINT := 1;
END_VAR
```

### KanLink_A19.typ - Global data types
```iecst
(********************************************************************
 * COPYRIGHT -- HP
 ********************************************************************
 * Package: KanLink_A7
 * File: KanLink_A7.typ
 * Author: treamsbottom
 * Created: January 28, 2013
 ********************************************************************
 * Data types of package KanLink_A7
 ********************************************************************)

TYPE
	IP_Type : 	STRUCT
		Area : UINT;
		Adr : UINT;
		CmdOpt : UINT;
		AdvMode : BOOL := FALSE;
		AdrAdvMode : STRING[15];
		CommID : USINT;
	END_STRUCT;
	KanOVClient_typ : 	STRUCT
		IP : ARRAY[0..HLKANLINK_MAX_CLIENTCONNS]OF IP_Type;
		Enable : BOOL;
		MaxConns : UINT;
		InfoReq : ARRAY[0..HLKANLINK_MAX_CLIENTCONNS]OF BatchInfo_typ;
		InfoResp : ARRAY[0..HLKANLINK_MAX_CLIENTCONNS]OF InfoResp_typ;
		StatusReg : ARRAY[0..HLKANLINK_MAX_CLIENTCONNS]OF UINT;
		IndexOffset : UINT;
		CANOffset : UINT; (**Can offset for CAN live index passed to Tview*)
	END_STRUCT;
	KanOVServer_typ : 	STRUCT
		IP : ARRAY[0..HLKANLINK_MAX_SERVERCONNS]OF IP_Type;
		Enable : BOOL;
		MaxConns : UINT;
		InfoResp : ARRAY[0..HLKANLINK_MAX_SERVERCONNS]OF KLresp1002_Info_typ;
		IndexOffset : UINT;
	END_STRUCT;
	KANServer_typ : 	STRUCT
		IP : ARRAY[0..HLKANLINK_MAX_SERVERCONNS]OF IP_Type;
		Enable : BOOL;
		MaxConns : UINT;
	END_STRUCT;
	KanLinkCon_Typ : 	STRUCT
		Server : KANServer_typ;
		Client : KANClient_typ;
		OverviewServer : KanOVServer_typ;
		OverviewClient : KanOVClient_typ;
		ErrorString : STRING[80];
		GlobalSettings : KAN_Settings;
	END_STRUCT;
	KANClient_typ : 	STRUCT
		IP : ARRAY[0..HLKANLINK_MAX_CLIENTCONNS]OF IP_Type;
		Enable : BOOL;
		MaxConns : UINT;
	END_STRUCT;
	BagNums_typ : 	STRUCT
		BagNums : ARRAY[0..6]OF UINT;
	END_STRUCT;
	KANBatch_typ : 	STRUCT
		BatchData : ARRAY[0..6]OF BatchData_typ;
	END_STRUCT;
	BatchInfo_typ : 	STRUCT
		wCntPositions : UINT;
		wNoOfPosition : ARRAY[0..HLKANLINK_MAX_OVERVIEW_DATA]OF UINT;
		wRes : UINT;
	END_STRUCT;
	InfoResp_typ : 	STRUCT
		BagNum : ARRAY[0..HLKANLINK_MAX_OVERVIEW_DATA]OF UINT;
	END_STRUCT;
	KAN_Settings : 	STRUCT
		UseBatchCode : BOOL;
		TransferProgramCode : BOOL; (**This puts the cat code in custom area and transfers the prg code to the m/c*)
		BatchCodeTyp : USINT;
		TransferProgin_bCustom : BOOL;
	END_STRUCT;
END_TYPE
```

### KanLink_A19.var - Global variables
```iecst
(********************************************************************
 * COPYRIGHT -- HP
 ********************************************************************
 * Package: KanLink_A2
 * File: KanLink_A2.var
 * Author: treamsbottom
 * Created: September 07, 2012
 ********************************************************************
 * Variables of package KanLink_A2
 ********************************************************************)
VAR
	Kanlink : KanLinkCon_Typ; (**Configuration parameters*)
	PTResp : ARRAY[0..HLKANLINK_MAX_CLIENTCONNS] OF KL_BTxf_typ; (**Client comm var*)
	PT100 : ARRAY[0..HLKANLINK_MAX_SERVERCONNS] OF KL_BTxf_typ; (**Server comm var*)
	Batch : ARRAY[0..HLKANLINK_MAX_SERVERCONNS] OF KANBatch_typ;
	STOverReq : ARRAY[0..HLKANLINK_MAX_CLIENTCONNS] OF KL_BI_typ; (*Overview Batch Info Server*)
	STOverResp : ARRAY[0..HLKANLINK_MAX_SERVERCONNS] OF KL_BI_typ; (*Overview Batch Info Client*)
END_VAR
```

### Program Logical/Standard/Kanlink/zz_KanlinkConfig (IEC, version 1.20.0) - *Configuration of Kanlink
